(* IEC 61131-3 sources: MotionTestBenchMaster/Logical/30_MC/Task/Cyclic03/MC_INTERFACE, 10 files *)

(* ---- HmiInterfaces.st ---- *)
ACTION HmiInterfaces:
	xAxisInVelocityControl	:= FALSE;

	IF VAR_Machine.iq_stParameter.i_uiAxisSelected >= CST_FillerSubModuleHmiStart AND VAR_Machine.iq_stParameter.i_uiAxisSelected <= CST_FillerSubModuleHmiStart + CST_LastFillerModuleAxis	THEN

		VAR_Machine.stFillerModule.iq_stParameters.i_uiAxisSelected	:= VAR_Machine.iq_stParameter.i_uiAxisSelected - CST_FillerSubModuleHmiStart;

		HMI_MC_GenericAxisData.uiDiagCode				:= VAR_Machine.stFillerModule.iq_astSubModuleAxis[VAR_Machine.stFillerModule.iq_stParameters.i_uiAxisSelected].iq_stStatus.q_stMainAxisStatus.q_stInfo.Diag.StatusID.Code;
		HMI_MC_GenericAxisData.iNextAx_Number;
		HMI_MC_GenericAxisData.iPrevAx_Number;
		HMI_MC_GenericAxisData.rEncoderTemperature		:= VAR_Machine.stFillerModule.iq_astSubModuleAxis[VAR_Machine.stFillerModule.iq_stParameters.i_uiAxisSelected].iq_stStatus.q_stMainAxisStatus.q_rEncoderTemperature;
		HMI_MC_GenericAxisData.rMaxTorque;
		HMI_MC_GenericAxisData.rMotorTemperature		:= VAR_Machine.stFillerModule.iq_astSubModuleAxis[VAR_Machine.stFillerModule.iq_stParameters.i_uiAxisSelected].iq_stStatus.q_stMainAxisStatus.q_rMotorTemperature;
		HMI_MC_GenericAxisData.rNextAx_Position_mm;
		HMI_MC_GenericAxisData.rPosition				:= LREAL_TO_REAL(VAR_Machine.stFillerModule.iq_astSubModuleAxis[VAR_Machine.stFillerModule.iq_stParameters.i_uiAxisSelected].iq_stStatus.q_stMainAxisStatus.q_lrPosition);
		HMI_MC_GenericAxisData.rPosition_mm				:= FC_DegreeToMm(CFG_MC.Mechanical.MachineStep, HMI_MC_GenericAxisData.rPosition, TRUE);

		HMI_MC_GenericAxisData.xMotorWithBrake			:= VAR_Machine.stFillerModule.iq_astSubModuleAxis[VAR_Machine.stFillerModule.iq_stParameters.i_uiAxisSelected].iq_stStatus.q_stMainAxisStatus.q_xMotorWithBrake;
		HMI_MC_GenericAxisData.xThirdPartMotor			:= VAR_Machine.stFillerModule.iq_astSubModuleAxis[VAR_Machine.stFillerModule.iq_stParameters.i_uiAxisSelected].iq_stStatus.q_stMainAxisStatus.q_xThirdPartyMotor;
		HMI_MC_GenericAxisData.xVelocityControl			:= VAR_Machine.stFillerModule.iq_astSubModuleAxis[VAR_Machine.stFillerModule.iq_stParameters.i_uiAxisSelected].iq_stStatus.q_stMainAxisStatus.q_xVelocityControl;
		HMI_MC_GenericAxisData.xInduction				:= VAR_Machine.stFillerModule.iq_astSubModuleAxis[VAR_Machine.stFillerModule.iq_stParameters.i_uiAxisSelected].iq_stStatus.q_stMainAxisStatus.q_xInduction;
		HMI_MC_GenericAxisData.rHomingOffset			:= VAR_Machine.stFillerModule.iq_astSubModuleAxis[VAR_Machine.stFillerModule.iq_stParameters.i_uiAxisSelected].iq_stStatus.q_stMainAxisStatus.q_rHomingOffset;

		HMI_MC_GenericAxisData.rTotalPhasingOffset		:= FC_DegreeToMm(CFG_MC.Mechanical.MachineStep,VAR_Machine.stFillerModule.iq_astSubModuleAxis[VAR_Machine.stFillerModule.iq_stParameters.i_uiAxisSelected].iq_stStatus.q_stMainAxisStatus.q_rTotalOffset, FALSE);

		HMI_MC_GenericAxisData.rLagError				:= FC_DegreeToMm(CFG_MC.Mechanical.MachineStep, VAR_Machine.stFillerModule.iq_astSubModuleAxis[VAR_Machine.stFillerModule.iq_stParameters.i_uiAxisSelected].iq_stStatus.q_stMainAxisStatus.q_rLagError, FALSE);

		HMI_MC_GenericAxisData.rPrevAx_Position_mm;
		HMI_MC_GenericAxisData.rTorque					:= LREAL_TO_REAL(VAR_Machine.stFillerModule.iq_astSubModuleAxis[VAR_Machine.stFillerModule.iq_stParameters.i_uiAxisSelected].iq_stStatus.q_stMainAxisStatus.q_lrTorque);
		HMI_MC_GenericAxisData.rVelocity				:= VAR_Machine.stFillerModule.iq_astSubModuleAxis[VAR_Machine.stFillerModule.iq_stParameters.i_uiAxisSelected].iq_stStatus.q_stMainAxisStatus.q_rVelocity * 10.0;
		HMI_MC_GenericAxisData.rSwitchValue;

		HMI_MC_GenericAxisData.xInitialized				:= VAR_Machine.stFillerModule.iq_astSubModuleAxis[VAR_Machine.stFillerModule.iq_stParameters.i_uiAxisSelected].iq_stStatus.q_stMainAxisStatus.q_xInitDone;

		xPhasingRunning									:= VAR_Machine.stFillerModule.iq_astSubModuleAxis[VAR_Machine.stFillerModule.iq_stParameters.i_uiAxisSelected].iq_stStatus.q_stMainAxisStatus.q_xPhasingRunning;

		IF HMI_MC_GenericAxisData.xInitialized THEN
			HMI_MC_GenericAxisData.xActive				:= VAR_Machine.stFillerModule.iq_astSubModuleAxis[VAR_Machine.stFillerModule.iq_stParameters.i_uiAxisSelected].iq_stStatus.q_stMainAxisStatus.q_xActive;
			HMI_MC_GenericAxisData.xBrakeReleased		:= VAR_Machine.stFillerModule.iq_astSubModuleAxis[VAR_Machine.stFillerModule.iq_stParameters.i_uiAxisSelected].iq_stStatus.q_stMainAxisStatus.q_xBrakeReleased;
			HMI_MC_GenericAxisData.xEnabled;
			HMI_MC_GenericAxisData.xFollowingError		:= VAR_Machine.stFillerModule.iq_astSubModuleAxis[VAR_Machine.stFillerModule.iq_stParameters.i_uiAxisSelected].iq_stStatus.q_stMainAxisStatus.q_xLagError;
			HMI_MC_GenericAxisData.xHomed				:= VAR_Machine.stFillerModule.iq_astSubModuleAxis[VAR_Machine.stFillerModule.iq_stParameters.i_uiAxisSelected].iq_stStatus.q_stMainAxisStatus.q_xIsHomed;
			HMI_MC_GenericAxisData.xInError				:= VAR_Machine.stFillerModule.iq_astSubModuleAxis[VAR_Machine.stFillerModule.iq_stParameters.i_uiAxisSelected].iq_stStatus.q_stMainAxisStatus.q_xError;
			HMI_MC_GenericAxisData.xInPosition			:= VAR_Machine.stFillerModule.iq_astSubModuleAxis[VAR_Machine.stFillerModule.iq_stParameters.i_uiAxisSelected].iq_stStatus.q_stMainAxisStatus.q_xInPosition;
			HMI_MC_GenericAxisData.xPowered				:= VAR_Machine.stFillerModule.iq_astSubModuleAxis[VAR_Machine.stFillerModule.iq_stParameters.i_uiAxisSelected].iq_stStatus.q_stMainAxisStatus.q_xPoweredOn;
			HMI_MC_GenericAxisData.xReal				:= VAR_Machine.stFillerModule.iq_astSubModuleAxis[VAR_Machine.stFillerModule.iq_stParameters.i_uiAxisSelected].iq_stStatus.q_stMainAxisStatus.q_xAxisReal;
			HMI_MC_GenericAxisData.xRunning				:= NOT VAR_Machine.stFillerModule.iq_astSubModuleAxis[VAR_Machine.stFillerModule.iq_stParameters.i_uiAxisSelected].iq_stStatus.q_stMainAxisStatus.q_xStopped;
			HMI_MC_GenericAxisData.xSynchro				:= VAR_Machine.stFillerModule.iq_astSubModuleAxis[VAR_Machine.stFillerModule.iq_stParameters.i_uiAxisSelected].iq_stStatus.q_stMainAxisStatus.q_xSynchronized;
			HMI_MC_GenericAxisData.xTorqueError			:= VAR_Machine.stFillerModule.iq_astSubModuleAxis[VAR_Machine.stFillerModule.iq_stParameters.i_uiAxisSelected].iq_stStatus.q_stMainAxisStatus.q_xTorqueError;
			HMI_MC_GenericAxisData.xHmiWait				:= FALSE;
		ELSE
			HMI_MC_GenericAxisData.xActive				:= FALSE;
			HMI_MC_GenericAxisData.xBrakeReleased		:= FALSE;
			HMI_MC_GenericAxisData.xEnabled;
			HMI_MC_GenericAxisData.xFollowingError		:= FALSE;
			HMI_MC_GenericAxisData.xHomed				:= FALSE;
			HMI_MC_GenericAxisData.xInError				:= FALSE;
			HMI_MC_GenericAxisData.xInPosition			:= FALSE;
			HMI_MC_GenericAxisData.xPowered				:= FALSE;
			HMI_MC_GenericAxisData.xReal				:= FALSE;
			HMI_MC_GenericAxisData.xRunning				:= FALSE;
			HMI_MC_GenericAxisData.xSynchro				:= FALSE;
			HMI_MC_GenericAxisData.xTorqueError			:= FALSE;
			HMI_MC_GenericAxisData.xHmiWait				:= TRUE;
		END_IF

		xAxisInVelocityControl	:= VAR_Machine.stFillerModule.iq_astSubModuleAxis[VAR_Machine.stFillerModule.iq_stParameters.i_uiAxisSelected].iq_stStatus.q_stMainAxisStatus.q_xVelocityControl;

	ELSIF VAR_Machine.iq_stParameter.i_uiAxisSelected >= CST_OutletSubModuleHmiStart AND VAR_Machine.iq_stParameter.i_uiAxisSelected <= CST_OutletSubModuleHmiStart + CST_LastOutletModuleAxis THEN

		VAR_Machine.stOutletModule.iq_stParameters.i_uiAxisSelected	:= VAR_Machine.iq_stParameter.i_uiAxisSelected - CST_OutletSubModuleHmiStart;

		HMI_MC_GenericAxisData.uiDiagCode				:= VAR_Machine.stOutletModule.iq_astSubModuleAxis[VAR_Machine.stOutletModule.iq_stParameters.i_uiAxisSelected].iq_stStatus.q_stMainAxisStatus.q_stInfo.Diag.StatusID.Code;
		HMI_MC_GenericAxisData.iNextAx_Number;
		HMI_MC_GenericAxisData.iPrevAx_Number;
		HMI_MC_GenericAxisData.rEncoderTemperature		:= VAR_Machine.stOutletModule.iq_astSubModuleAxis[VAR_Machine.stOutletModule.iq_stParameters.i_uiAxisSelected].iq_stStatus.q_stMainAxisStatus.q_rEncoderTemperature;
		HMI_MC_GenericAxisData.rMaxTorque;
		HMI_MC_GenericAxisData.rLagError				:= FC_DegreeToMm(CFG_MC.Mechanical.MachineStep, VAR_Machine.stOutletModule.iq_astSubModuleAxis[VAR_Machine.stOutletModule.iq_stParameters.i_uiAxisSelected].iq_stStatus.q_stMainAxisStatus.q_rLagError, FALSE);

		HMI_MC_GenericAxisData.xMotorWithBrake			:= VAR_Machine.stOutletModule.iq_astSubModuleAxis[VAR_Machine.stOutletModule.iq_stParameters.i_uiAxisSelected].iq_stStatus.q_stMainAxisStatus.q_xMotorWithBrake;
		HMI_MC_GenericAxisData.xThirdPartMotor			:= VAR_Machine.stOutletModule.iq_astSubModuleAxis[VAR_Machine.stOutletModule.iq_stParameters.i_uiAxisSelected].iq_stStatus.q_stMainAxisStatus.q_xThirdPartyMotor;
		HMI_MC_GenericAxisData.xVelocityControl			:= VAR_Machine.stOutletModule.iq_astSubModuleAxis[VAR_Machine.stOutletModule.iq_stParameters.i_uiAxisSelected].iq_stStatus.q_stMainAxisStatus.q_xVelocityControl;
		HMI_MC_GenericAxisData.xInduction				:= VAR_Machine.stOutletModule.iq_astSubModuleAxis[VAR_Machine.stOutletModule.iq_stParameters.i_uiAxisSelected].iq_stStatus.q_stMainAxisStatus.q_xInduction;
		HMI_MC_GenericAxisData.rHomingOffset			:= VAR_Machine.stOutletModule.iq_astSubModuleAxis[VAR_Machine.stOutletModule.iq_stParameters.i_uiAxisSelected].iq_stStatus.q_stMainAxisStatus.q_rHomingOffset;

		HMI_MC_GenericAxisData.rMotorTemperature		:= VAR_Machine.stOutletModule.iq_astSubModuleAxis[VAR_Machine.stOutletModule.iq_stParameters.i_uiAxisSelected].iq_stStatus.q_stMainAxisStatus.q_rMotorTemperature;
		HMI_MC_GenericAxisData.rNextAx_Position_mm;
		HMI_MC_GenericAxisData.rPosition				:= LREAL_TO_REAL(VAR_Machine.stOutletModule.iq_astSubModuleAxis[VAR_Machine.stOutletModule.iq_stParameters.i_uiAxisSelected].iq_stStatus.q_stMainAxisStatus.q_lrPosition);
		HMI_MC_GenericAxisData.rPosition_mm				:= FC_DegreeToMm(CFG_MC.Mechanical.MachineStep, HMI_MC_GenericAxisData.rPosition, TRUE);

		HMI_MC_GenericAxisData.rPrevAx_Position_mm;
		HMI_MC_GenericAxisData.rTorque					:= LREAL_TO_REAL(VAR_Machine.stOutletModule.iq_astSubModuleAxis[VAR_Machine.stOutletModule.iq_stParameters.i_uiAxisSelected].iq_stStatus.q_stMainAxisStatus.q_lrTorque);
		HMI_MC_GenericAxisData.rVelocity				:= VAR_Machine.stOutletModule.iq_astSubModuleAxis[VAR_Machine.stOutletModule.iq_stParameters.i_uiAxisSelected].iq_stStatus.q_stMainAxisStatus.q_rVelocity * 10.0;
		HMI_MC_GenericAxisData.rSwitchValue;

		HMI_MC_GenericAxisData.rTotalPhasingOffset		:= FC_DegreeToMm(CFG_MC.Mechanical.MachineStep,VAR_Machine.stOutletModule.iq_astSubModuleAxis[VAR_Machine.stOutletModule.iq_stParameters.i_uiAxisSelected].iq_stStatus.q_stMainAxisStatus.q_rTotalOffset,FALSE);

		HMI_MC_GenericAxisData.xInitialized				:= VAR_Machine.stOutletModule.iq_astSubModuleAxis[VAR_Machine.stOutletModule.iq_stParameters.i_uiAxisSelected].iq_stStatus.q_stMainAxisStatus.q_xInitDone;

		xPhasingRunning									:= VAR_Machine.stOutletModule.iq_astSubModuleAxis[VAR_Machine.stOutletModule.iq_stParameters.i_uiAxisSelected].iq_stStatus.q_stMainAxisStatus.q_xPhasingRunning;

		IF HMI_MC_GenericAxisData.xInitialized THEN
			HMI_MC_GenericAxisData.xActive				:= VAR_Machine.stOutletModule.iq_astSubModuleAxis[VAR_Machine.stOutletModule.iq_stParameters.i_uiAxisSelected].iq_stStatus.q_stMainAxisStatus.q_xActive;
			HMI_MC_GenericAxisData.xBrakeReleased		:= VAR_Machine.stOutletModule.iq_astSubModuleAxis[VAR_Machine.stOutletModule.iq_stParameters.i_uiAxisSelected].iq_stStatus.q_stMainAxisStatus.q_xBrakeReleased;
			HMI_MC_GenericAxisData.xEnabled;
			HMI_MC_GenericAxisData.xFollowingError		:= VAR_Machine.stOutletModule.iq_astSubModuleAxis[VAR_Machine.stOutletModule.iq_stParameters.i_uiAxisSelected].iq_stStatus.q_stMainAxisStatus.q_xLagError;
			HMI_MC_GenericAxisData.xHomed				:= VAR_Machine.stOutletModule.iq_astSubModuleAxis[VAR_Machine.stOutletModule.iq_stParameters.i_uiAxisSelected].iq_stStatus.q_stMainAxisStatus.q_xIsHomed;
			HMI_MC_GenericAxisData.xInError				:= VAR_Machine.stOutletModule.iq_astSubModuleAxis[VAR_Machine.stOutletModule.iq_stParameters.i_uiAxisSelected].iq_stStatus.q_stMainAxisStatus.q_xError;
			HMI_MC_GenericAxisData.xInPosition			:= VAR_Machine.stOutletModule.iq_astSubModuleAxis[VAR_Machine.stOutletModule.iq_stParameters.i_uiAxisSelected].iq_stStatus.q_stMainAxisStatus.q_xInPosition;
			HMI_MC_GenericAxisData.xPowered				:= VAR_Machine.stOutletModule.iq_astSubModuleAxis[VAR_Machine.stOutletModule.iq_stParameters.i_uiAxisSelected].iq_stStatus.q_stMainAxisStatus.q_xPoweredOn;
			HMI_MC_GenericAxisData.xReal				:= VAR_Machine.stOutletModule.iq_astSubModuleAxis[VAR_Machine.stOutletModule.iq_stParameters.i_uiAxisSelected].iq_stStatus.q_stMainAxisStatus.q_xAxisReal;
			HMI_MC_GenericAxisData.xRunning				:= NOT VAR_Machine.stOutletModule.iq_astSubModuleAxis[VAR_Machine.stOutletModule.iq_stParameters.i_uiAxisSelected].iq_stStatus.q_stMainAxisStatus.q_xStopped;
			HMI_MC_GenericAxisData.xSynchro				:= VAR_Machine.stOutletModule.iq_astSubModuleAxis[VAR_Machine.stOutletModule.iq_stParameters.i_uiAxisSelected].iq_stStatus.q_stMainAxisStatus.q_xSynchronized;
			HMI_MC_GenericAxisData.xTorqueError			:= VAR_Machine.stOutletModule.iq_astSubModuleAxis[VAR_Machine.stOutletModule.iq_stParameters.i_uiAxisSelected].iq_stStatus.q_stMainAxisStatus.q_xTorqueError;
			HMI_MC_GenericAxisData.xHmiWait				:= FALSE;
		ELSE
			HMI_MC_GenericAxisData.xActive				:= FALSE;
			HMI_MC_GenericAxisData.xBrakeReleased		:= FALSE;
			HMI_MC_GenericAxisData.xEnabled;
			HMI_MC_GenericAxisData.xFollowingError		:= FALSE;
			HMI_MC_GenericAxisData.xHomed				:= FALSE;
			HMI_MC_GenericAxisData.xInError				:= FALSE;
			HMI_MC_GenericAxisData.xInPosition			:= FALSE;
			HMI_MC_GenericAxisData.xPowered				:= FALSE;
			HMI_MC_GenericAxisData.xReal				:= FALSE;
			HMI_MC_GenericAxisData.xRunning				:= FALSE;
			HMI_MC_GenericAxisData.xSynchro				:= FALSE;
			HMI_MC_GenericAxisData.xTorqueError			:= FALSE;
			HMI_MC_GenericAxisData.xHmiWait				:= TRUE;
		END_IF

		xAxisInVelocityControl	:= VAR_Machine.stOutletModule.iq_astSubModuleAxis[VAR_Machine.stOutletModule.iq_stParameters.i_uiAxisSelected].iq_stStatus.q_stMainAxisStatus.q_xVelocityControl;

	ELSIF VAR_Machine.iq_stParameter.i_uiAxisSelected >= CST_InletSubModuleHmiStart AND VAR_Machine.iq_stParameter.i_uiAxisSelected <= CST_InletSubModuleHmiStart + CST_LastInletModuleAxis THEN

		VAR_Machine.stInletModule.iq_stParameters.i_uiAxisSelected	:= VAR_Machine.iq_stParameter.i_uiAxisSelected - CST_InletSubModuleHmiStart;

		HMI_MC_GenericAxisData.uiDiagCode				:= VAR_Machine.stInletModule.iq_astSubModuleAxis[VAR_Machine.stInletModule.iq_stParameters.i_uiAxisSelected].iq_stStatus.q_stMainAxisStatus.q_stInfo.Diag.StatusID.Code;
		HMI_MC_GenericAxisData.iNextAx_Number;
		HMI_MC_GenericAxisData.iPrevAx_Number;
		HMI_MC_GenericAxisData.rEncoderTemperature		:= VAR_Machine.stInletModule.iq_astSubModuleAxis[VAR_Machine.stInletModule.iq_stParameters.i_uiAxisSelected].iq_stStatus.q_stMainAxisStatus.q_rEncoderTemperature;
		HMI_MC_GenericAxisData.rMaxTorque;
		HMI_MC_GenericAxisData.rLagError				:= FC_DegreeToMm(CFG_MC.Mechanical.MachineStep, VAR_Machine.stInletModule.iq_astSubModuleAxis[VAR_Machine.stInletModule.iq_stParameters.i_uiAxisSelected].iq_stStatus.q_stMainAxisStatus.q_rLagError, FALSE);

		HMI_MC_GenericAxisData.xMotorWithBrake			:= VAR_Machine.stInletModule.iq_astSubModuleAxis[VAR_Machine.stInletModule.iq_stParameters.i_uiAxisSelected].iq_stStatus.q_stMainAxisStatus.q_xMotorWithBrake;
		HMI_MC_GenericAxisData.xThirdPartMotor			:= VAR_Machine.stInletModule.iq_astSubModuleAxis[VAR_Machine.stInletModule.iq_stParameters.i_uiAxisSelected].iq_stStatus.q_stMainAxisStatus.q_xThirdPartyMotor;
		HMI_MC_GenericAxisData.xVelocityControl			:= VAR_Machine.stInletModule.iq_astSubModuleAxis[VAR_Machine.stInletModule.iq_stParameters.i_uiAxisSelected].iq_stStatus.q_stMainAxisStatus.q_xVelocityControl;
		HMI_MC_GenericAxisData.xInduction				:= VAR_Machine.stInletModule.iq_astSubModuleAxis[VAR_Machine.stInletModule.iq_stParameters.i_uiAxisSelected].iq_stStatus.q_stMainAxisStatus.q_xInduction;
		HMI_MC_GenericAxisData.rHomingOffset			:= VAR_Machine.stInletModule.iq_astSubModuleAxis[VAR_Machine.stInletModule.iq_stParameters.i_uiAxisSelected].iq_stStatus.q_stMainAxisStatus.q_rHomingOffset;

		HMI_MC_GenericAxisData.rMotorTemperature		:= VAR_Machine.stInletModule.iq_astSubModuleAxis[VAR_Machine.stInletModule.iq_stParameters.i_uiAxisSelected].iq_stStatus.q_stMainAxisStatus.q_rMotorTemperature;
		HMI_MC_GenericAxisData.rNextAx_Position_mm;
		HMI_MC_GenericAxisData.rPosition				:= LREAL_TO_REAL(VAR_Machine.stInletModule.iq_astSubModuleAxis[VAR_Machine.stInletModule.iq_stParameters.i_uiAxisSelected].iq_stStatus.q_stMainAxisStatus.q_lrPosition);
		HMI_MC_GenericAxisData.rPosition_mm				:= FC_DegreeToMm(CFG_MC.Mechanical.MachineStep, HMI_MC_GenericAxisData.rPosition, TRUE);

		HMI_MC_GenericAxisData.rPrevAx_Position_mm;
		HMI_MC_GenericAxisData.rTorque					:= LREAL_TO_REAL(VAR_Machine.stInletModule.iq_astSubModuleAxis[VAR_Machine.stInletModule.iq_stParameters.i_uiAxisSelected].iq_stStatus.q_stMainAxisStatus.q_lrTorque);
		HMI_MC_GenericAxisData.rVelocity				:= VAR_Machine.stInletModule.iq_astSubModuleAxis[VAR_Machine.stInletModule.iq_stParameters.i_uiAxisSelected].iq_stStatus.q_stMainAxisStatus.q_rVelocity * 10.0;
		HMI_MC_GenericAxisData.rSwitchValue;

		HMI_MC_GenericAxisData.rTotalPhasingOffset		:= FC_DegreeToMm(CFG_MC.Mechanical.MachineStep,VAR_Machine.stInletModule.iq_astSubModuleAxis[VAR_Machine.stInletModule.iq_stParameters.i_uiAxisSelected].iq_stStatus.q_stMainAxisStatus.q_rTotalOffset,FALSE);

		HMI_MC_GenericAxisData.xInitialized				:= VAR_Machine.stInletModule.iq_astSubModuleAxis[VAR_Machine.stInletModule.iq_stParameters.i_uiAxisSelected].iq_stStatus.q_stMainAxisStatus.q_xInitDone;

		xPhasingRunning									:= VAR_Machine.stInletModule.iq_astSubModuleAxis[VAR_Machine.stInletModule.iq_stParameters.i_uiAxisSelected].iq_stStatus.q_stMainAxisStatus.q_xPhasingRunning;

		IF HMI_MC_GenericAxisData.xInitialized THEN
			HMI_MC_GenericAxisData.xActive				:= VAR_Machine.stInletModule.iq_astSubModuleAxis[VAR_Machine.stInletModule.iq_stParameters.i_uiAxisSelected].iq_stStatus.q_stMainAxisStatus.q_xActive;
			HMI_MC_GenericAxisData.xBrakeReleased		:= VAR_Machine.stInletModule.iq_astSubModuleAxis[VAR_Machine.stInletModule.iq_stParameters.i_uiAxisSelected].iq_stStatus.q_stMainAxisStatus.q_xBrakeReleased;
			HMI_MC_GenericAxisData.xEnabled;
			HMI_MC_GenericAxisData.xFollowingError		:= VAR_Machine.stInletModule.iq_astSubModuleAxis[VAR_Machine.stInletModule.iq_stParameters.i_uiAxisSelected].iq_stStatus.q_stMainAxisStatus.q_xLagError;
			HMI_MC_GenericAxisData.xHomed				:= VAR_Machine.stInletModule.iq_astSubModuleAxis[VAR_Machine.stInletModule.iq_stParameters.i_uiAxisSelected].iq_stStatus.q_stMainAxisStatus.q_xIsHomed;
			HMI_MC_GenericAxisData.xInError				:= VAR_Machine.stInletModule.iq_astSubModuleAxis[VAR_Machine.stInletModule.iq_stParameters.i_uiAxisSelected].iq_stStatus.q_stMainAxisStatus.q_xError;
			HMI_MC_GenericAxisData.xInPosition			:= VAR_Machine.stInletModule.iq_astSubModuleAxis[VAR_Machine.stInletModule.iq_stParameters.i_uiAxisSelected].iq_stStatus.q_stMainAxisStatus.q_xInPosition;
			HMI_MC_GenericAxisData.xPowered				:= VAR_Machine.stInletModule.iq_astSubModuleAxis[VAR_Machine.stInletModule.iq_stParameters.i_uiAxisSelected].iq_stStatus.q_stMainAxisStatus.q_xPoweredOn;
			HMI_MC_GenericAxisData.xReal				:= VAR_Machine.stInletModule.iq_astSubModuleAxis[VAR_Machine.stInletModule.iq_stParameters.i_uiAxisSelected].iq_stStatus.q_stMainAxisStatus.q_xAxisReal;
			HMI_MC_GenericAxisData.xRunning				:= NOT VAR_Machine.stInletModule.iq_astSubModuleAxis[VAR_Machine.stInletModule.iq_stParameters.i_uiAxisSelected].iq_stStatus.q_stMainAxisStatus.q_xStopped;
			HMI_MC_GenericAxisData.xSynchro				:= VAR_Machine.stInletModule.iq_astSubModuleAxis[VAR_Machine.stInletModule.iq_stParameters.i_uiAxisSelected].iq_stStatus.q_stMainAxisStatus.q_xSynchronized;
			HMI_MC_GenericAxisData.xTorqueError			:= VAR_Machine.stInletModule.iq_astSubModuleAxis[VAR_Machine.stInletModule.iq_stParameters.i_uiAxisSelected].iq_stStatus.q_stMainAxisStatus.q_xTorqueError;
			HMI_MC_GenericAxisData.xHmiWait				:= FALSE;
		ELSE
			HMI_MC_GenericAxisData.xActive				:= FALSE;
			HMI_MC_GenericAxisData.xBrakeReleased		:= FALSE;
			HMI_MC_GenericAxisData.xEnabled;
			HMI_MC_GenericAxisData.xFollowingError		:= FALSE;
			HMI_MC_GenericAxisData.xHomed				:= FALSE;
			HMI_MC_GenericAxisData.xInError				:= FALSE;
			HMI_MC_GenericAxisData.xInPosition			:= FALSE;
			HMI_MC_GenericAxisData.xPowered				:= FALSE;
			HMI_MC_GenericAxisData.xReal				:= FALSE;
			HMI_MC_GenericAxisData.xRunning				:= FALSE;
			HMI_MC_GenericAxisData.xSynchro				:= FALSE;
			HMI_MC_GenericAxisData.xTorqueError			:= FALSE;
			HMI_MC_GenericAxisData.xHmiWait				:= TRUE;
		END_IF

		xAxisInVelocityControl	:= VAR_Machine.stInletModule.iq_astSubModuleAxis[VAR_Machine.stInletModule.iq_stParameters.i_uiAxisSelected].iq_stStatus.q_stMainAxisStatus.q_xVelocityControl;

	ELSIF VAR_Machine.iq_stParameter.i_uiAxisSelected = CST_MachinePhasingOffset THEN

		VAR_Machine.stMasterModule.iq_stParameters.i_uiAxisSelected	:=	VAR_Machine.iq_stParameter.i_uiAxisSelected;

		HMI_MC_GenericAxisData.uiDiagCode				:= VAR_Machine.stMasterModule.iq_astSubModuleAxis[CST_MachineMasterAxis].iq_stStatus.q_stMainAxisStatus.q_stInfo.Diag.StatusID.Code;
		HMI_MC_GenericAxisData.rLagError				:= FC_DegreeToMm(CFG_MC.Mechanical.MachineStep, VAR_Machine.stMasterModule.iq_astSubModuleAxis[CST_MachineMasterAxis].iq_stStatus.q_stMainAxisStatus.q_rLagError,FALSE);

		HMI_MC_GenericAxisData.xMotorWithBrake			:= VAR_Machine.stMasterModule.iq_astSubModuleAxis[CST_MachineMasterAxis].iq_stStatus.q_stMainAxisStatus.q_xMotorWithBrake;
		HMI_MC_GenericAxisData.xThirdPartMotor			:= VAR_Machine.stMasterModule.iq_astSubModuleAxis[CST_MachineMasterAxis].iq_stStatus.q_stMainAxisStatus.q_xThirdPartyMotor;
		HMI_MC_GenericAxisData.xVelocityControl			:= VAR_Machine.stMasterModule.iq_astSubModuleAxis[CST_MachineMasterAxis].iq_stStatus.q_stMainAxisStatus.q_xVelocityControl;
		HMI_MC_GenericAxisData.xInduction				:= VAR_Machine.stMasterModule.iq_astSubModuleAxis[CST_MachineMasterAxis].iq_stStatus.q_stMainAxisStatus.q_xInduction;
		HMI_MC_GenericAxisData.rHomingOffset			:= VAR_Machine.stMasterModule.iq_astSubModuleAxis[CST_MachineMasterAxis].iq_stStatus.q_stMainAxisStatus.q_rHomingOffset;

		HMI_MC_GenericAxisData.rPosition				:= LREAL_TO_REAL(VAR_Machine.stMasterModule.iq_astSubModuleAxis[CST_MachineMasterAxis].iq_stStatus.q_stMainAxisStatus.q_lrPosition);
		HMI_MC_GenericAxisData.rPosition_mm				:= FC_DegreeToMm(CFG_MC.Mechanical.MachineStep,HMI_MC_GenericAxisData.rPosition,TRUE);

		HMI_MC_GenericAxisData.rVelocity				:= VAR_Machine.stMasterModule.iq_astSubModuleAxis[CST_MachineMasterAxis].iq_stStatus.q_stMainAxisStatus.q_rVelocity * 10.0;

		HMI_MC_GenericAxisData.rTotalPhasingOffset		:= FC_DegreeToMm(CFG_MC.Mechanical.MachineStep,VAR_Machine.stMasterModule.iq_astSubModuleAxis[CST_MachineMasterAxis].iq_stStatus.q_stMainAxisStatus.q_rTotalOffset,FALSE);

		HMI_MC_GenericAxisData.xInitialized				:= VAR_Machine.stMasterModule.iq_astSubModuleAxis[CST_MachineMasterAxis].iq_stStatus.q_stMainAxisStatus.q_xInitDone;

		xPhasingRunning									:= VAR_Machine.stMasterModule.iq_astSubModuleAxis[CST_MachineMasterAxis].iq_stStatus.q_stMainAxisStatus.q_xPhasingRunning;

		IF HMI_MC_GenericAxisData.xInitialized THEN
			HMI_MC_GenericAxisData.xActive				:= VAR_Machine.stMasterModule.iq_astSubModuleAxis[CST_MachineMasterAxis].iq_stStatus.q_stMainAxisStatus.q_xActive;
			HMI_MC_GenericAxisData.xBrakeReleased		:= FALSE;
			HMI_MC_GenericAxisData.xEnabled;
			HMI_MC_GenericAxisData.xFollowingError		:= FALSE;
			HMI_MC_GenericAxisData.xHomed				:= FALSE;
			HMI_MC_GenericAxisData.xInError				:= VAR_Machine.stMasterModule.iq_astSubModuleAxis[CST_MachineMasterAxis].iq_stStatus.q_stMainAxisStatus.q_xError;
			HMI_MC_GenericAxisData.xInPosition			:= VAR_Machine.stMasterModule.iq_astSubModuleAxis[CST_MachineMasterAxis].iq_stStatus.q_stMainAxisStatus.q_xInPosition;
			HMI_MC_GenericAxisData.xPowered				:= FALSE;
			HMI_MC_GenericAxisData.xReal				:= FALSE;
			HMI_MC_GenericAxisData.xRunning				:= FALSE;
			HMI_MC_GenericAxisData.xSynchro				:= VAR_Machine.stMasterModule.iq_astSubModuleAxis[CST_MachineMasterAxis].iq_stStatus.q_stMainAxisStatus.q_xSynchronized;
			HMI_MC_GenericAxisData.xTorqueError			:= FALSE;
			HMI_MC_GenericAxisData.xHmiWait				:= FALSE;
		ELSE
			HMI_MC_GenericAxisData.xActive				:= FALSE;
			HMI_MC_GenericAxisData.xBrakeReleased		:= FALSE;
			HMI_MC_GenericAxisData.xEnabled;
			HMI_MC_GenericAxisData.xFollowingError		:= FALSE;
			HMI_MC_GenericAxisData.xHomed				:= FALSE;
			HMI_MC_GenericAxisData.xInError				:= FALSE;
			HMI_MC_GenericAxisData.xInPosition			:= FALSE;
			HMI_MC_GenericAxisData.xPowered				:= FALSE;
			HMI_MC_GenericAxisData.xReal				:= FALSE;
			HMI_MC_GenericAxisData.xRunning				:= FALSE;
			HMI_MC_GenericAxisData.xSynchro				:= FALSE;
			HMI_MC_GenericAxisData.xTorqueError			:= FALSE;
			HMI_MC_GenericAxisData.xHmiWait				:= TRUE;
		END_IF

		xAxisInVelocityControl	:=	 VAR_Machine.stMasterModule.iq_astSubModuleAxis[CST_MachineMasterAxis].iq_stStatus.q_stMainAxisStatus.q_xVelocityControl;
	END_IF

	CASE VAR_Machine.iq_stParameter.i_uiAxisSelected OF
		99:
			HMI_MC_GenericAxisData.usiHmiName	:= 99; //V4.A.A.1.6.13

		105:
			HMI_MC_GenericAxisData.usiHmiName	:= CFG_MC.Axes.Filler.In[10].HmiNameId;

		106:
			HMI_MC_GenericAxisData.usiHmiName	:= CFG_MC.Axes.Filler.In[9].HmiNameId;

		107:
			HMI_MC_GenericAxisData.usiHmiName	:= CFG_MC.Axes.Filler.In[8].HmiNameId;

		108:
			HMI_MC_GenericAxisData.usiHmiName	:= CFG_MC.Axes.Filler.In[7].HmiNameId;

		109:
			HMI_MC_GenericAxisData.usiHmiName	:= CFG_MC.Axes.Filler.In[6].HmiNameId;

		110:
			HMI_MC_GenericAxisData.usiHmiName	:= CFG_MC.Axes.Filler.In[5].HmiNameId;

		111:
			HMI_MC_GenericAxisData.usiHmiName	:= CFG_MC.Axes.Filler.In[4].HmiNameId;

		112:
			HMI_MC_GenericAxisData.usiHmiName	:= CFG_MC.Axes.Filler.In[3].HmiNameId;

		113:
			HMI_MC_GenericAxisData.usiHmiName	:= CFG_MC.Axes.Filler.In[2].HmiNameId;

		114:
			HMI_MC_GenericAxisData.usiHmiName	:= CFG_MC.Axes.Filler.In[1].HmiNameId;

		115:
			HMI_MC_GenericAxisData.usiHmiName	:= CFG_MC.Axes.Filler.Main.HmiNameId;

		116:
			HMI_MC_GenericAxisData.usiHmiName	:= CFG_MC.Axes.Filler.Out[1].HmiNameId;

		117:
			HMI_MC_GenericAxisData.usiHmiName	:= CFG_MC.Axes.Filler.Out[2].HmiNameId;

		118:
			HMI_MC_GenericAxisData.usiHmiName	:= CFG_MC.Axes.Filler.Out[3].HmiNameId;

		119:
			HMI_MC_GenericAxisData.usiHmiName	:= CFG_MC.Axes.Filler.Out[4].HmiNameId;

		120:
			HMI_MC_GenericAxisData.usiHmiName	:= CFG_MC.Axes.Filler.Out[5].HmiNameId;

		121:
			HMI_MC_GenericAxisData.usiHmiName	:= CFG_MC.Axes.Filler.Out[6].HmiNameId;

		211:
			HMI_MC_GenericAxisData.usiHmiName	:= CFG_MC.Axes.Inlet.In[4].HmiNameId;

		212:
			HMI_MC_GenericAxisData.usiHmiName	:= CFG_MC.Axes.Inlet.In[3].HmiNameId;

		213:
			HMI_MC_GenericAxisData.usiHmiName	:= CFG_MC.Axes.Inlet.In[2].HmiNameId;

		214:
			HMI_MC_GenericAxisData.usiHmiName	:= CFG_MC.Axes.Inlet.In[1].HmiNameId;

		215:
			HMI_MC_GenericAxisData.usiHmiName	:= CFG_MC.Axes.Inlet.Main.HmiNameId;

		216:
			HMI_MC_GenericAxisData.usiHmiName	:= CFG_MC.Axes.Inlet.Out[1].HmiNameId;

		217:
			HMI_MC_GenericAxisData.usiHmiName	:= CFG_MC.Axes.Inlet.Out[2].HmiNameId;

		218:
			HMI_MC_GenericAxisData.usiHmiName	:= CFG_MC.Axes.Inlet.Out[3].HmiNameId;

		219:
			HMI_MC_GenericAxisData.usiHmiName	:= CFG_MC.Axes.Inlet.Out[4].HmiNameId;

		311:
			HMI_MC_GenericAxisData.usiHmiName	:= CFG_MC.Axes.Outlet.In[4].HmiNameId;

		312:
			HMI_MC_GenericAxisData.usiHmiName	:= CFG_MC.Axes.Outlet.In[3].HmiNameId;

		313:
			HMI_MC_GenericAxisData.usiHmiName	:= CFG_MC.Axes.Outlet.In[2].HmiNameId;

		314:
			HMI_MC_GenericAxisData.usiHmiName	:= CFG_MC.Axes.Outlet.In[1].HmiNameId;

		315:
			HMI_MC_GenericAxisData.usiHmiName	:= CFG_MC.Axes.Outlet.Main.HmiNameId;

		316:
			HMI_MC_GenericAxisData.usiHmiName	:= CFG_MC.Axes.Outlet.Out[1].HmiNameId;

		317:
			HMI_MC_GenericAxisData.usiHmiName	:= CFG_MC.Axes.Outlet.Out[2].HmiNameId;

		318:
			HMI_MC_GenericAxisData.usiHmiName	:= CFG_MC.Axes.Outlet.Out[3].HmiNameId;

		319:
			HMI_MC_GenericAxisData.usiHmiName	:= CFG_MC.Axes.Outlet.Out[4].HmiNameId;
		ELSE
			HMI_MC_GenericAxisData.usiHmiName		:= 0;
	END_CASE

	HMI_MC_AxisPresent;

	//Transfer Wheel - Encoder Diagnostic
	HMI_MC_EncoderDiagnostic.Present 	:= CFG_MC.Generic.SyncroPar.ExternalEncoder;
	HMI_MC_EncoderDiagnostic.ModuleOK 	:= MC_InputOutput.Network.Machine.Commands.MasterEncoderPositionValid;
	HMI_MC_EncoderDiagnostic.Value 		:= ITC_Motion_ExtEnc;
END_ACTION

(* ---- HmiInterfacesNew.st ---- *)
ACTION HmiInterfacesNew:
	xAxisInVelocityControl	:= FALSE;

	IF VAR_Machine.iq_stParameter.i_uiAxisSelected >= CST_FillerSubModuleHmiStart AND VAR_Machine.iq_stParameter.i_uiAxisSelected <= CST_FillerSubModuleHmiStart + CST_LastFillerModuleAxis	THEN
		VAR_Machine.stFillerModule.iq_stParameters.i_uiAxisSelected	:= VAR_Machine.iq_stParameter.i_uiAxisSelected - CST_FillerSubModuleHmiStart;
	ELSIF VAR_Machine.iq_stParameter.i_uiAxisSelected >= CST_OutletSubModuleHmiStart AND VAR_Machine.iq_stParameter.i_uiAxisSelected <= CST_OutletSubModuleHmiStart + CST_LastOutletModuleAxis THEN
		VAR_Machine.stOutletModule.iq_stParameters.i_uiAxisSelected	:= VAR_Machine.iq_stParameter.i_uiAxisSelected - CST_OutletSubModuleHmiStart;
	ELSIF VAR_Machine.iq_stParameter.i_uiAxisSelected >= CST_InletSubModuleHmiStart AND VAR_Machine.iq_stParameter.i_uiAxisSelected <= CST_InletSubModuleHmiStart + CST_LastInletModuleAxis THEN
		VAR_Machine.stInletModule.iq_stParameters.i_uiAxisSelected	:= VAR_Machine.iq_stParameter.i_uiAxisSelected - CST_InletSubModuleHmiStart;
	ELSIF VAR_Machine.iq_stParameter.i_uiAxisSelected = CST_MachinePhasingOffset THEN
		VAR_Machine.stMasterModule.iq_stParameters.i_uiAxisSelected	:=	VAR_Machine.iq_stParameter.i_uiAxisSelected;
	END_IF
////////////////////////////////////////////////

		HMI_MC_GenericAxisDataNew[1].uiDiagCode				:= VAR_Machine.stMasterModule.iq_astSubModuleAxis[CST_MachineMasterAxis].iq_stStatus.q_stMainAxisStatus.q_stInfo.Diag.StatusID.Code;
		HMI_MC_GenericAxisDataNew[1].rLagError				:= FC_DegreeToMm(CFG_MC.Mechanical.MachineStep, VAR_Machine.stMasterModule.iq_astSubModuleAxis[CST_MachineMasterAxis].iq_stStatus.q_stMainAxisStatus.q_rLagError,FALSE);

		HMI_MC_GenericAxisDataNew[1].xMotorWithBrake		:= VAR_Machine.stMasterModule.iq_astSubModuleAxis[CST_MachineMasterAxis].iq_stStatus.q_stMainAxisStatus.q_xMotorWithBrake;
		HMI_MC_GenericAxisDataNew[1].xThirdPartMotor		:= VAR_Machine.stMasterModule.iq_astSubModuleAxis[CST_MachineMasterAxis].iq_stStatus.q_stMainAxisStatus.q_xThirdPartyMotor;
		HMI_MC_GenericAxisDataNew[1].xVelocityControl		:= VAR_Machine.stMasterModule.iq_astSubModuleAxis[CST_MachineMasterAxis].iq_stStatus.q_stMainAxisStatus.q_xVelocityControl;
		HMI_MC_GenericAxisDataNew[1].xInduction				:= VAR_Machine.stMasterModule.iq_astSubModuleAxis[CST_MachineMasterAxis].iq_stStatus.q_stMainAxisStatus.q_xInduction;
		HMI_MC_GenericAxisDataNew[1].rHomingOffset			:= VAR_Machine.stMasterModule.iq_astSubModuleAxis[CST_MachineMasterAxis].iq_stStatus.q_stMainAxisStatus.q_rHomingOffset;

		HMI_MC_GenericAxisDataNew[1].rPosition				:= LREAL_TO_REAL(VAR_Machine.stMasterModule.iq_astSubModuleAxis[CST_MachineMasterAxis].iq_stStatus.q_stMainAxisStatus.q_lrPosition);
		HMI_MC_GenericAxisDataNew[1].rPosition_mm			:= FC_DegreeToMm(CFG_MC.Mechanical.MachineStep,HMI_MC_GenericAxisDataNew[1].rPosition,TRUE);//V1.7.2

		HMI_MC_GenericAxisDataNew[1].rVelocity				:= VAR_Machine.stMasterModule.iq_astSubModuleAxis[CST_MachineMasterAxis].iq_stStatus.q_stMainAxisStatus.q_rVelocity * 10.0;

		HMI_MC_GenericAxisDataNew[1].rTotalPhasingOffset	:= FC_DegreeToMm(CFG_MC.Mechanical.MachineStep,VAR_Machine.stMasterModule.iq_astSubModuleAxis[CST_MachineMasterAxis].iq_stStatus.q_stMainAxisStatus.q_rTotalOffset,FALSE);

		HMI_MC_GenericAxisDataNew[1].xInitialized			:= VAR_Machine.stMasterModule.iq_astSubModuleAxis[CST_MachineMasterAxis].iq_stStatus.q_stMainAxisStatus.q_xInitDone;

		xPhasingRunning									:= VAR_Machine.stMasterModule.iq_astSubModuleAxis[CST_MachineMasterAxis].iq_stStatus.q_stMainAxisStatus.q_xPhasingRunning;

		IF HMI_MC_GenericAxisDataNew[1].xInitialized THEN
			HMI_MC_GenericAxisDataNew[1].xActive				:= VAR_Machine.stMasterModule.iq_astSubModuleAxis[CST_MachineMasterAxis].iq_stStatus.q_stMainAxisStatus.q_xActive;
			HMI_MC_GenericAxisDataNew[1].xBrakeReleased		:= FALSE;
			HMI_MC_GenericAxisDataNew[1].xEnabled;
			HMI_MC_GenericAxisDataNew[1].xFollowingError		:= FALSE;
			HMI_MC_GenericAxisDataNew[1].xHomed				:= FALSE;
			HMI_MC_GenericAxisDataNew[1].xInError				:= VAR_Machine.stMasterModule.iq_astSubModuleAxis[CST_MachineMasterAxis].iq_stStatus.q_stMainAxisStatus.q_xError;
			HMI_MC_GenericAxisDataNew[1].xInPosition			:= VAR_Machine.stMasterModule.iq_astSubModuleAxis[CST_MachineMasterAxis].iq_stStatus.q_stMainAxisStatus.q_xInPosition;
			HMI_MC_GenericAxisDataNew[1].xPowered				:= FALSE;
			HMI_MC_GenericAxisDataNew[1].xReal				:= FALSE;
			HMI_MC_GenericAxisDataNew[1].xRunning				:= FALSE;
			HMI_MC_GenericAxisDataNew[1].xSynchro				:= VAR_Machine.stMasterModule.iq_astSubModuleAxis[CST_MachineMasterAxis].iq_stStatus.q_stMainAxisStatus.q_xSynchronized;
			HMI_MC_GenericAxisDataNew[1].xTorqueError			:= FALSE;
//			HMI_MC_GenericAxisDataNew[1].xHmiWait				:= FALSE;//V1.7.2
		ELSE
			HMI_MC_GenericAxisDataNew[1].xActive				:= FALSE;
			HMI_MC_GenericAxisDataNew[1].xBrakeReleased		:= FALSE;
			HMI_MC_GenericAxisDataNew[1].xEnabled;
			HMI_MC_GenericAxisDataNew[1].xFollowingError		:= FALSE;
			HMI_MC_GenericAxisDataNew[1].xHomed				:= FALSE;
			HMI_MC_GenericAxisDataNew[1].xInError				:= FALSE;
			HMI_MC_GenericAxisDataNew[1].xInPosition			:= FALSE;
			HMI_MC_GenericAxisDataNew[1].xPowered				:= FALSE;
			HMI_MC_GenericAxisDataNew[1].xReal				:= FALSE;
			HMI_MC_GenericAxisDataNew[1].xRunning				:= FALSE;
			HMI_MC_GenericAxisDataNew[1].xSynchro				:= FALSE;
			HMI_MC_GenericAxisDataNew[1].xTorqueError			:= FALSE;
//			HMI_MC_GenericAxisDataNew[1].xHmiWait				:= TRUE;//v1.7.2
		END_IF

	FOR HMI_AxisIndex := 1 TO 13 DO
		//Inlet Axis Motor
		IF HMI_MC_GenericAxisDataNew[HMI_AxisIndex].uiAxisID >= CST_InletSubModuleHmiStart AND HMI_MC_GenericAxisDataNew[HMI_AxisIndex].uiAxisID <= CST_InletSubModuleHmiStart + CST_LastInletModuleAxis THEN

			HMI_MC_GenericAxisDataNew[HMI_AxisIndex].uiDiagCode				:= VAR_Machine.stInletModule.iq_astSubModuleAxis[HMI_MC_GenericAxisDataNew[HMI_AxisIndex].uiAxisID-CST_InletSubModuleHmiStart].iq_stStatus.q_stMainAxisStatus.q_stInfo.Diag.StatusID.Code;
			HMI_MC_GenericAxisDataNew[HMI_AxisIndex].iNextAx_Number;
			HMI_MC_GenericAxisDataNew[HMI_AxisIndex].iPrevAx_Number;
			HMI_MC_GenericAxisDataNew[HMI_AxisIndex].rEncoderTemperature		:= VAR_Machine.stInletModule.iq_astSubModuleAxis[HMI_MC_GenericAxisDataNew[HMI_AxisIndex].uiAxisID-CST_InletSubModuleHmiStart].iq_stStatus.q_stMainAxisStatus.q_rEncoderTemperature;
			HMI_MC_GenericAxisDataNew[HMI_AxisIndex].rMaxTorque;
			HMI_MC_GenericAxisDataNew[HMI_AxisIndex].rLagError				:= FC_DegreeToMm(CFG_MC.Mechanical.MachineStep, VAR_Machine.stInletModule.iq_astSubModuleAxis[HMI_MC_GenericAxisDataNew[HMI_AxisIndex].uiAxisID-CST_InletSubModuleHmiStart].iq_stStatus.q_stMainAxisStatus.q_rLagError, FALSE);

			HMI_MC_GenericAxisDataNew[HMI_AxisIndex].xMotorWithBrake			:= VAR_Machine.stInletModule.iq_astSubModuleAxis[HMI_MC_GenericAxisDataNew[HMI_AxisIndex].uiAxisID-CST_InletSubModuleHmiStart].iq_stStatus.q_stMainAxisStatus.q_xMotorWithBrake;
			HMI_MC_GenericAxisDataNew[HMI_AxisIndex].xThirdPartMotor			:= VAR_Machine.stInletModule.iq_astSubModuleAxis[HMI_MC_GenericAxisDataNew[HMI_AxisIndex].uiAxisID-CST_InletSubModuleHmiStart].iq_stStatus.q_stMainAxisStatus.q_xThirdPartyMotor;
			HMI_MC_GenericAxisDataNew[HMI_AxisIndex].xVelocityControl			:= VAR_Machine.stInletModule.iq_astSubModuleAxis[HMI_MC_GenericAxisDataNew[HMI_AxisIndex].uiAxisID-CST_InletSubModuleHmiStart].iq_stStatus.q_stMainAxisStatus.q_xVelocityControl;
			HMI_MC_GenericAxisDataNew[HMI_AxisIndex].xInduction				:= VAR_Machine.stInletModule.iq_astSubModuleAxis[HMI_MC_GenericAxisDataNew[HMI_AxisIndex].uiAxisID-CST_InletSubModuleHmiStart].iq_stStatus.q_stMainAxisStatus.q_xInduction;
			HMI_MC_GenericAxisDataNew[HMI_AxisIndex].rHomingOffset			:= VAR_Machine.stInletModule.iq_astSubModuleAxis[HMI_MC_GenericAxisDataNew[HMI_AxisIndex].uiAxisID-CST_InletSubModuleHmiStart].iq_stStatus.q_stMainAxisStatus.q_rHomingOffset;

			HMI_MC_GenericAxisDataNew[HMI_AxisIndex].rMotorTemperature		:= VAR_Machine.stInletModule.iq_astSubModuleAxis[HMI_MC_GenericAxisDataNew[HMI_AxisIndex].uiAxisID-CST_InletSubModuleHmiStart].iq_stStatus.q_stMainAxisStatus.q_rMotorTemperature;
			HMI_MC_GenericAxisDataNew[HMI_AxisIndex].rNextAx_Position_mm;
			HMI_MC_GenericAxisDataNew[HMI_AxisIndex].rPosition				:= LREAL_TO_REAL(VAR_Machine.stInletModule.iq_astSubModuleAxis[HMI_MC_GenericAxisDataNew[HMI_AxisIndex].uiAxisID-CST_InletSubModuleHmiStart].iq_stStatus.q_stMainAxisStatus.q_lrPosition);
			HMI_MC_GenericAxisDataNew[HMI_AxisIndex].rPosition_mm			:= FC_DegreeToMm(CFG_MC.Mechanical.MachineStep,HMI_MC_GenericAxisDataNew[HMI_AxisIndex].rPosition,TRUE);//v1.7.2

			HMI_MC_GenericAxisDataNew[HMI_AxisIndex].rPrevAx_Position_mm;
			HMI_MC_GenericAxisDataNew[HMI_AxisIndex].rTorque					:= LREAL_TO_REAL(VAR_Machine.stInletModule.iq_astSubModuleAxis[HMI_MC_GenericAxisDataNew[HMI_AxisIndex].uiAxisID-CST_InletSubModuleHmiStart].iq_stStatus.q_stMainAxisStatus.q_lrTorque);
			HMI_MC_GenericAxisDataNew[HMI_AxisIndex].rVelocity				:= VAR_Machine.stInletModule.iq_astSubModuleAxis[HMI_MC_GenericAxisDataNew[HMI_AxisIndex].uiAxisID-CST_InletSubModuleHmiStart].iq_stStatus.q_stMainAxisStatus.q_rVelocity * 10.0;
			HMI_MC_GenericAxisDataNew[HMI_AxisIndex].rSwitchValue;

			HMI_MC_GenericAxisDataNew[HMI_AxisIndex].rTotalPhasingOffset		:= FC_DegreeToMm(CFG_MC.Mechanical.MachineStep,VAR_Machine.stInletModule.iq_astSubModuleAxis[HMI_MC_GenericAxisDataNew[HMI_AxisIndex].uiAxisID-CST_InletSubModuleHmiStart].iq_stStatus.q_stMainAxisStatus.q_rTotalOffset,FALSE);

			HMI_MC_GenericAxisDataNew[HMI_AxisIndex].xInitialized				:= VAR_Machine.stInletModule.iq_astSubModuleAxis[HMI_MC_GenericAxisDataNew[HMI_AxisIndex].uiAxisID-CST_InletSubModuleHmiStart].iq_stStatus.q_stMainAxisStatus.q_xInitDone;

			xPhasingRunning									:= VAR_Machine.stInletModule.iq_astSubModuleAxis[HMI_MC_GenericAxisDataNew[HMI_AxisIndex].uiAxisID-CST_InletSubModuleHmiStart].iq_stStatus.q_stMainAxisStatus.q_xPhasingRunning;

			IF HMI_MC_GenericAxisDataNew[HMI_AxisIndex].xInitialized THEN
				HMI_MC_GenericAxisDataNew[HMI_AxisIndex].xActive				:= VAR_Machine.stInletModule.iq_astSubModuleAxis[HMI_MC_GenericAxisDataNew[HMI_AxisIndex].uiAxisID-CST_InletSubModuleHmiStart].iq_stStatus.q_stMainAxisStatus.q_xActive;
				HMI_MC_GenericAxisDataNew[HMI_AxisIndex].xBrakeReleased		:= VAR_Machine.stInletModule.iq_astSubModuleAxis[HMI_MC_GenericAxisDataNew[HMI_AxisIndex].uiAxisID-CST_InletSubModuleHmiStart].iq_stStatus.q_stMainAxisStatus.q_xBrakeReleased;
				HMI_MC_GenericAxisDataNew[HMI_AxisIndex].xEnabled;
				HMI_MC_GenericAxisDataNew[HMI_AxisIndex].xFollowingError		:= VAR_Machine.stInletModule.iq_astSubModuleAxis[HMI_MC_GenericAxisDataNew[HMI_AxisIndex].uiAxisID-CST_InletSubModuleHmiStart].iq_stStatus.q_stMainAxisStatus.q_xLagError;
				HMI_MC_GenericAxisDataNew[HMI_AxisIndex].xHomed				:= VAR_Machine.stInletModule.iq_astSubModuleAxis[HMI_MC_GenericAxisDataNew[HMI_AxisIndex].uiAxisID-CST_InletSubModuleHmiStart].iq_stStatus.q_stMainAxisStatus.q_xIsHomed;
				HMI_MC_GenericAxisDataNew[HMI_AxisIndex].xInError				:= VAR_Machine.stInletModule.iq_astSubModuleAxis[HMI_MC_GenericAxisDataNew[HMI_AxisIndex].uiAxisID-CST_InletSubModuleHmiStart].iq_stStatus.q_stMainAxisStatus.q_xError;
				HMI_MC_GenericAxisDataNew[HMI_AxisIndex].xInPosition			:= VAR_Machine.stInletModule.iq_astSubModuleAxis[HMI_MC_GenericAxisDataNew[HMI_AxisIndex].uiAxisID-CST_InletSubModuleHmiStart].iq_stStatus.q_stMainAxisStatus.q_xInPosition;
				HMI_MC_GenericAxisDataNew[HMI_AxisIndex].xPowered				:= VAR_Machine.stInletModule.iq_astSubModuleAxis[HMI_MC_GenericAxisDataNew[HMI_AxisIndex].uiAxisID-CST_InletSubModuleHmiStart].iq_stStatus.q_stMainAxisStatus.q_xPoweredOn;
				HMI_MC_GenericAxisDataNew[HMI_AxisIndex].xReal				:= VAR_Machine.stInletModule.iq_astSubModuleAxis[HMI_MC_GenericAxisDataNew[HMI_AxisIndex].uiAxisID-CST_InletSubModuleHmiStart].iq_stStatus.q_stMainAxisStatus.q_xAxisReal;
				HMI_MC_GenericAxisDataNew[HMI_AxisIndex].xRunning				:= NOT VAR_Machine.stInletModule.iq_astSubModuleAxis[HMI_MC_GenericAxisDataNew[HMI_AxisIndex].uiAxisID-CST_InletSubModuleHmiStart].iq_stStatus.q_stMainAxisStatus.q_xStopped;
				HMI_MC_GenericAxisDataNew[HMI_AxisIndex].xSynchro				:= VAR_Machine.stInletModule.iq_astSubModuleAxis[HMI_MC_GenericAxisDataNew[HMI_AxisIndex].uiAxisID-CST_InletSubModuleHmiStart].iq_stStatus.q_stMainAxisStatus.q_xSynchronized;
				HMI_MC_GenericAxisDataNew[HMI_AxisIndex].xTorqueError			:= VAR_Machine.stInletModule.iq_astSubModuleAxis[HMI_MC_GenericAxisDataNew[HMI_AxisIndex].uiAxisID-CST_InletSubModuleHmiStart].iq_stStatus.q_stMainAxisStatus.q_xTorqueError;
				//HMI_MC_GenericAxisDataNew[HMI_AxisIndex].xHmiWait				:= FALSE;//v1.7.2
			ELSE
				HMI_MC_GenericAxisDataNew[HMI_AxisIndex].xActive				:= FALSE;
				HMI_MC_GenericAxisDataNew[HMI_AxisIndex].xBrakeReleased		:= FALSE;
				HMI_MC_GenericAxisDataNew[HMI_AxisIndex].xEnabled;
				HMI_MC_GenericAxisDataNew[HMI_AxisIndex].xFollowingError		:= FALSE;
				HMI_MC_GenericAxisDataNew[HMI_AxisIndex].xHomed					:= FALSE;
				HMI_MC_GenericAxisDataNew[HMI_AxisIndex].xInError				:= FALSE;
				HMI_MC_GenericAxisDataNew[HMI_AxisIndex].xInPosition			:= FALSE;
				HMI_MC_GenericAxisDataNew[HMI_AxisIndex].xPowered				:= FALSE;
				HMI_MC_GenericAxisDataNew[HMI_AxisIndex].xReal					:= FALSE;
				HMI_MC_GenericAxisDataNew[HMI_AxisIndex].xRunning				:= FALSE;
				HMI_MC_GenericAxisDataNew[HMI_AxisIndex].xSynchro				:= FALSE;
				HMI_MC_GenericAxisDataNew[HMI_AxisIndex].xTorqueError			:= FALSE;
//				HMI_MC_GenericAxisDataNew[HMI_AxisIndex].xHmiWait				:= TRUE;//v1.7.2
			END_IF
			xAxisInVelocityControl	:= VAR_Machine.stInletModule.iq_astSubModuleAxis[HMI_MC_GenericAxisDataNew[HMI_AxisIndex].uiAxisID-CST_InletSubModuleHmiStart].iq_stStatus.q_stMainAxisStatus.q_xVelocityControl;
		//Filler Module
		ELSIF HMI_MC_GenericAxisDataNew[HMI_AxisIndex].uiAxisID >= CST_FillerSubModuleHmiStart AND HMI_MC_GenericAxisDataNew[HMI_AxisIndex].uiAxisID <= CST_FillerSubModuleHmiStart + CST_LastFillerModuleAxis THEN
			HMI_MC_GenericAxisDataNew[HMI_AxisIndex].uiDiagCode				:= VAR_Machine.stFillerModule.iq_astSubModuleAxis[HMI_MC_GenericAxisDataNew[HMI_AxisIndex].uiAxisID-CST_FillerSubModuleHmiStart].iq_stStatus.q_stMainAxisStatus.q_stInfo.Diag.StatusID.Code;
			HMI_MC_GenericAxisDataNew[HMI_AxisIndex].iNextAx_Number;
			HMI_MC_GenericAxisDataNew[HMI_AxisIndex].iPrevAx_Number;
			HMI_MC_GenericAxisDataNew[HMI_AxisIndex].rEncoderTemperature		:= VAR_Machine.stFillerModule.iq_astSubModuleAxis[HMI_MC_GenericAxisDataNew[HMI_AxisIndex].uiAxisID-CST_FillerSubModuleHmiStart].iq_stStatus.q_stMainAxisStatus.q_rEncoderTemperature;
			HMI_MC_GenericAxisDataNew[HMI_AxisIndex].rMaxTorque;
			HMI_MC_GenericAxisDataNew[HMI_AxisIndex].rMotorTemperature		:= VAR_Machine.stFillerModule.iq_astSubModuleAxis[HMI_MC_GenericAxisDataNew[HMI_AxisIndex].uiAxisID-CST_FillerSubModuleHmiStart].iq_stStatus.q_stMainAxisStatus.q_rMotorTemperature;
			HMI_MC_GenericAxisDataNew[HMI_AxisIndex].rNextAx_Position_mm;
			HMI_MC_GenericAxisDataNew[HMI_AxisIndex].rPosition				:= LREAL_TO_REAL(VAR_Machine.stFillerModule.iq_astSubModuleAxis[HMI_MC_GenericAxisDataNew[HMI_AxisIndex].uiAxisID-CST_FillerSubModuleHmiStart].iq_stStatus.q_stMainAxisStatus.q_lrPosition);
			HMI_MC_GenericAxisDataNew[HMI_AxisIndex].rPosition_mm			:= FC_DegreeToMm(CFG_MC.Mechanical.MachineStep,HMI_MC_GenericAxisDataNew[HMI_AxisIndex].rPosition,TRUE);//v1.7.2

			HMI_MC_GenericAxisDataNew[HMI_AxisIndex].xMotorWithBrake			:= VAR_Machine.stFillerModule.iq_astSubModuleAxis[HMI_MC_GenericAxisDataNew[HMI_AxisIndex].uiAxisID-CST_FillerSubModuleHmiStart].iq_stStatus.q_stMainAxisStatus.q_xMotorWithBrake;
			HMI_MC_GenericAxisDataNew[HMI_AxisIndex].xThirdPartMotor			:= VAR_Machine.stFillerModule.iq_astSubModuleAxis[HMI_MC_GenericAxisDataNew[HMI_AxisIndex].uiAxisID-CST_FillerSubModuleHmiStart].iq_stStatus.q_stMainAxisStatus.q_xThirdPartyMotor;
			HMI_MC_GenericAxisDataNew[HMI_AxisIndex].xVelocityControl			:= VAR_Machine.stFillerModule.iq_astSubModuleAxis[HMI_MC_GenericAxisDataNew[HMI_AxisIndex].uiAxisID-CST_FillerSubModuleHmiStart].iq_stStatus.q_stMainAxisStatus.q_xVelocityControl;
			HMI_MC_GenericAxisDataNew[HMI_AxisIndex].xInduction				:= VAR_Machine.stFillerModule.iq_astSubModuleAxis[HMI_MC_GenericAxisDataNew[HMI_AxisIndex].uiAxisID-CST_FillerSubModuleHmiStart].iq_stStatus.q_stMainAxisStatus.q_xInduction;
			HMI_MC_GenericAxisDataNew[HMI_AxisIndex].rHomingOffset			:= VAR_Machine.stFillerModule.iq_astSubModuleAxis[HMI_MC_GenericAxisDataNew[HMI_AxisIndex].uiAxisID-CST_FillerSubModuleHmiStart].iq_stStatus.q_stMainAxisStatus.q_rHomingOffset;

			HMI_MC_GenericAxisDataNew[HMI_AxisIndex].rTotalPhasingOffset		:= FC_DegreeToMm(CFG_MC.Mechanical.MachineStep,VAR_Machine.stFillerModule.iq_astSubModuleAxis[HMI_MC_GenericAxisDataNew[HMI_AxisIndex].uiAxisID-CST_FillerSubModuleHmiStart].iq_stStatus.q_stMainAxisStatus.q_rTotalOffset, FALSE);

			HMI_MC_GenericAxisDataNew[HMI_AxisIndex].rLagError				:= FC_DegreeToMm(CFG_MC.Mechanical.MachineStep, VAR_Machine.stFillerModule.iq_astSubModuleAxis[HMI_MC_GenericAxisDataNew[HMI_AxisIndex].uiAxisID-CST_FillerSubModuleHmiStart].iq_stStatus.q_stMainAxisStatus.q_rLagError, FALSE);

			HMI_MC_GenericAxisDataNew[HMI_AxisIndex].rPrevAx_Position_mm;
			HMI_MC_GenericAxisDataNew[HMI_AxisIndex].rTorque					:= LREAL_TO_REAL(VAR_Machine.stFillerModule.iq_astSubModuleAxis[HMI_MC_GenericAxisDataNew[HMI_AxisIndex].uiAxisID-CST_FillerSubModuleHmiStart].iq_stStatus.q_stMainAxisStatus.q_lrTorque);
			HMI_MC_GenericAxisDataNew[HMI_AxisIndex].rVelocity				:= VAR_Machine.stFillerModule.iq_astSubModuleAxis[HMI_MC_GenericAxisDataNew[HMI_AxisIndex].uiAxisID-CST_FillerSubModuleHmiStart].iq_stStatus.q_stMainAxisStatus.q_rVelocity * 10.0;
			HMI_MC_GenericAxisDataNew[HMI_AxisIndex].rSwitchValue;

			HMI_MC_GenericAxisDataNew[HMI_AxisIndex].xInitialized				:= VAR_Machine.stFillerModule.iq_astSubModuleAxis[HMI_MC_GenericAxisDataNew[HMI_AxisIndex].uiAxisID-CST_FillerSubModuleHmiStart].iq_stStatus.q_stMainAxisStatus.q_xInitDone;

			xPhasingRunning									:= VAR_Machine.stFillerModule.iq_astSubModuleAxis[HMI_MC_GenericAxisDataNew[HMI_AxisIndex].uiAxisID-CST_FillerSubModuleHmiStart].iq_stStatus.q_stMainAxisStatus.q_xPhasingRunning;

			IF HMI_MC_GenericAxisDataNew[HMI_AxisIndex].xInitialized THEN
				HMI_MC_GenericAxisDataNew[HMI_AxisIndex].xActive				:= VAR_Machine.stFillerModule.iq_astSubModuleAxis[HMI_MC_GenericAxisDataNew[HMI_AxisIndex].uiAxisID-CST_FillerSubModuleHmiStart].iq_stStatus.q_stMainAxisStatus.q_xActive;
				HMI_MC_GenericAxisDataNew[HMI_AxisIndex].xBrakeReleased		:= VAR_Machine.stFillerModule.iq_astSubModuleAxis[HMI_MC_GenericAxisDataNew[HMI_AxisIndex].uiAxisID-CST_FillerSubModuleHmiStart].iq_stStatus.q_stMainAxisStatus.q_xBrakeReleased;
				HMI_MC_GenericAxisDataNew[HMI_AxisIndex].xEnabled;
				HMI_MC_GenericAxisDataNew[HMI_AxisIndex].xFollowingError		:= VAR_Machine.stFillerModule.iq_astSubModuleAxis[HMI_MC_GenericAxisDataNew[HMI_AxisIndex].uiAxisID-CST_FillerSubModuleHmiStart].iq_stStatus.q_stMainAxisStatus.q_xLagError;
				HMI_MC_GenericAxisDataNew[HMI_AxisIndex].xHomed				:= VAR_Machine.stFillerModule.iq_astSubModuleAxis[HMI_MC_GenericAxisDataNew[HMI_AxisIndex].uiAxisID-CST_FillerSubModuleHmiStart].iq_stStatus.q_stMainAxisStatus.q_xIsHomed;
				HMI_MC_GenericAxisDataNew[HMI_AxisIndex].xInError				:= VAR_Machine.stFillerModule.iq_astSubModuleAxis[HMI_MC_GenericAxisDataNew[HMI_AxisIndex].uiAxisID-CST_FillerSubModuleHmiStart].iq_stStatus.q_stMainAxisStatus.q_xError;
				HMI_MC_GenericAxisDataNew[HMI_AxisIndex].xInPosition			:= VAR_Machine.stFillerModule.iq_astSubModuleAxis[HMI_MC_GenericAxisDataNew[HMI_AxisIndex].uiAxisID-CST_FillerSubModuleHmiStart].iq_stStatus.q_stMainAxisStatus.q_xInPosition;
				HMI_MC_GenericAxisDataNew[HMI_AxisIndex].xPowered				:= VAR_Machine.stFillerModule.iq_astSubModuleAxis[HMI_MC_GenericAxisDataNew[HMI_AxisIndex].uiAxisID-CST_FillerSubModuleHmiStart].iq_stStatus.q_stMainAxisStatus.q_xPoweredOn;
				HMI_MC_GenericAxisDataNew[HMI_AxisIndex].xReal				:= VAR_Machine.stFillerModule.iq_astSubModuleAxis[HMI_MC_GenericAxisDataNew[HMI_AxisIndex].uiAxisID-CST_FillerSubModuleHmiStart].iq_stStatus.q_stMainAxisStatus.q_xAxisReal;
				HMI_MC_GenericAxisDataNew[HMI_AxisIndex].xRunning				:= NOT VAR_Machine.stFillerModule.iq_astSubModuleAxis[HMI_MC_GenericAxisDataNew[HMI_AxisIndex].uiAxisID-CST_FillerSubModuleHmiStart].iq_stStatus.q_stMainAxisStatus.q_xStopped;
				HMI_MC_GenericAxisDataNew[HMI_AxisIndex].xSynchro				:= VAR_Machine.stFillerModule.iq_astSubModuleAxis[HMI_MC_GenericAxisDataNew[HMI_AxisIndex].uiAxisID-CST_FillerSubModuleHmiStart].iq_stStatus.q_stMainAxisStatus.q_xSynchronized;
				HMI_MC_GenericAxisDataNew[HMI_AxisIndex].xTorqueError			:= VAR_Machine.stFillerModule.iq_astSubModuleAxis[HMI_MC_GenericAxisDataNew[HMI_AxisIndex].uiAxisID-CST_FillerSubModuleHmiStart].iq_stStatus.q_stMainAxisStatus.q_xTorqueError;
				//HMI_MC_GenericAxisDataNew[HMI_AxisIndex].xHmiWait				:= FALSE;//v1.7.2
			ELSE
				HMI_MC_GenericAxisDataNew[HMI_AxisIndex].xActive				:= FALSE;
				HMI_MC_GenericAxisDataNew[HMI_AxisIndex].xBrakeReleased		:= FALSE;
				HMI_MC_GenericAxisDataNew[HMI_AxisIndex].xEnabled;
				HMI_MC_GenericAxisDataNew[HMI_AxisIndex].xFollowingError		:= FALSE;
				HMI_MC_GenericAxisDataNew[HMI_AxisIndex].xHomed				:= FALSE;
				HMI_MC_GenericAxisDataNew[HMI_AxisIndex].xInError				:= FALSE;
				HMI_MC_GenericAxisDataNew[HMI_AxisIndex].xInPosition			:= FALSE;
				HMI_MC_GenericAxisDataNew[HMI_AxisIndex].xPowered				:= FALSE;
				HMI_MC_GenericAxisDataNew[HMI_AxisIndex].xReal				:= FALSE;
				HMI_MC_GenericAxisDataNew[HMI_AxisIndex].xRunning				:= FALSE;
				HMI_MC_GenericAxisDataNew[HMI_AxisIndex].xSynchro				:= FALSE;
				HMI_MC_GenericAxisDataNew[HMI_AxisIndex].xTorqueError			:= FALSE;
				//HMI_MC_GenericAxisDataNew[HMI_AxisIndex].xHmiWait				:= TRUE;//v1.7.2
			END_IF

			xAxisInVelocityControl	:= VAR_Machine.stFillerModule.iq_astSubModuleAxis[HMI_MC_GenericAxisDataNew[HMI_AxisIndex].uiAxisID-CST_FillerSubModuleHmiStart].iq_stStatus.q_stMainAxisStatus.q_xVelocityControl;
		//Outlet Module
		ELSIF HMI_MC_GenericAxisDataNew[HMI_AxisIndex].uiAxisID >= CST_OutletSubModuleHmiStart AND HMI_MC_GenericAxisDataNew[HMI_AxisIndex].uiAxisID <= CST_OutletSubModuleHmiStart + CST_LastOutletModuleAxis THEN
			HMI_MC_GenericAxisDataNew[HMI_AxisIndex].uiDiagCode					:= VAR_Machine.stOutletModule.iq_astSubModuleAxis[HMI_MC_GenericAxisDataNew[HMI_AxisIndex].uiAxisID - CST_OutletSubModuleHmiStart].iq_stStatus.q_stMainAxisStatus.q_stInfo.Diag.StatusID.Code;
			HMI_MC_GenericAxisDataNew[HMI_AxisIndex].iNextAx_Number;
			HMI_MC_GenericAxisDataNew[HMI_AxisIndex].iPrevAx_Number;
			HMI_MC_GenericAxisDataNew[HMI_AxisIndex].rEncoderTemperature		:= VAR_Machine.stOutletModule.iq_astSubModuleAxis[HMI_MC_GenericAxisDataNew[HMI_AxisIndex].uiAxisID - CST_OutletSubModuleHmiStart].iq_stStatus.q_stMainAxisStatus.q_rEncoderTemperature;
			HMI_MC_GenericAxisDataNew[HMI_AxisIndex].rMaxTorque;
			HMI_MC_GenericAxisDataNew[HMI_AxisIndex].rLagError					:= FC_DegreeToMm(CFG_MC.Mechanical.MachineStep, VAR_Machine.stOutletModule.iq_astSubModuleAxis[HMI_MC_GenericAxisDataNew[HMI_AxisIndex].uiAxisID - CST_OutletSubModuleHmiStart].iq_stStatus.q_stMainAxisStatus.q_rLagError, FALSE);

			HMI_MC_GenericAxisDataNew[HMI_AxisIndex].xMotorWithBrake			:= VAR_Machine.stOutletModule.iq_astSubModuleAxis[HMI_MC_GenericAxisDataNew[HMI_AxisIndex].uiAxisID - CST_OutletSubModuleHmiStart].iq_stStatus.q_stMainAxisStatus.q_xMotorWithBrake;
			HMI_MC_GenericAxisDataNew[HMI_AxisIndex].xThirdPartMotor			:= VAR_Machine.stOutletModule.iq_astSubModuleAxis[HMI_MC_GenericAxisDataNew[HMI_AxisIndex].uiAxisID - CST_OutletSubModuleHmiStart].iq_stStatus.q_stMainAxisStatus.q_xThirdPartyMotor;
			HMI_MC_GenericAxisDataNew[HMI_AxisIndex].xVelocityControl			:= VAR_Machine.stOutletModule.iq_astSubModuleAxis[HMI_MC_GenericAxisDataNew[HMI_AxisIndex].uiAxisID - CST_OutletSubModuleHmiStart].iq_stStatus.q_stMainAxisStatus.q_xVelocityControl;
			HMI_MC_GenericAxisDataNew[HMI_AxisIndex].xInduction					:= VAR_Machine.stOutletModule.iq_astSubModuleAxis[HMI_MC_GenericAxisDataNew[HMI_AxisIndex].uiAxisID - CST_OutletSubModuleHmiStart].iq_stStatus.q_stMainAxisStatus.q_xInduction;
			HMI_MC_GenericAxisDataNew[HMI_AxisIndex].rHomingOffset				:= VAR_Machine.stOutletModule.iq_astSubModuleAxis[HMI_MC_GenericAxisDataNew[HMI_AxisIndex].uiAxisID - CST_OutletSubModuleHmiStart].iq_stStatus.q_stMainAxisStatus.q_rHomingOffset;

			HMI_MC_GenericAxisDataNew[HMI_AxisIndex].rMotorTemperature			:= VAR_Machine.stOutletModule.iq_astSubModuleAxis[HMI_MC_GenericAxisDataNew[HMI_AxisIndex].uiAxisID - CST_OutletSubModuleHmiStart].iq_stStatus.q_stMainAxisStatus.q_rMotorTemperature;
			HMI_MC_GenericAxisDataNew[HMI_AxisIndex].rNextAx_Position_mm;
			HMI_MC_GenericAxisDataNew[HMI_AxisIndex].rPosition					:= LREAL_TO_REAL(VAR_Machine.stOutletModule.iq_astSubModuleAxis[HMI_MC_GenericAxisDataNew[HMI_AxisIndex].uiAxisID - CST_OutletSubModuleHmiStart].iq_stStatus.q_stMainAxisStatus.q_lrPosition);
			HMI_MC_GenericAxisDataNew[HMI_AxisIndex].rPosition_mm				:= FC_DegreeToMm(CFG_MC.Mechanical.MachineStep,HMI_MC_GenericAxisDataNew[HMI_AxisIndex].rPosition,TRUE);//v1.7.2

			HMI_MC_GenericAxisDataNew[HMI_AxisIndex].rPrevAx_Position_mm;
			HMI_MC_GenericAxisDataNew[HMI_AxisIndex].rTorque					:= LREAL_TO_REAL(VAR_Machine.stOutletModule.iq_astSubModuleAxis[HMI_MC_GenericAxisDataNew[HMI_AxisIndex].uiAxisID - CST_OutletSubModuleHmiStart].iq_stStatus.q_stMainAxisStatus.q_lrTorque);
			HMI_MC_GenericAxisDataNew[HMI_AxisIndex].rVelocity					:= VAR_Machine.stOutletModule.iq_astSubModuleAxis[HMI_MC_GenericAxisDataNew[HMI_AxisIndex].uiAxisID - CST_OutletSubModuleHmiStart].iq_stStatus.q_stMainAxisStatus.q_rVelocity * 10.0;
			HMI_MC_GenericAxisDataNew[HMI_AxisIndex].rSwitchValue;

			HMI_MC_GenericAxisDataNew[HMI_AxisIndex].rTotalPhasingOffset		:= FC_DegreeToMm(CFG_MC.Mechanical.MachineStep,VAR_Machine.stOutletModule.iq_astSubModuleAxis[HMI_MC_GenericAxisDataNew[HMI_AxisIndex].uiAxisID - CST_OutletSubModuleHmiStart].iq_stStatus.q_stMainAxisStatus.q_rTotalOffset,FALSE);

			HMI_MC_GenericAxisDataNew[HMI_AxisIndex].xInitialized				:= VAR_Machine.stOutletModule.iq_astSubModuleAxis[HMI_MC_GenericAxisDataNew[HMI_AxisIndex].uiAxisID - CST_OutletSubModuleHmiStart].iq_stStatus.q_stMainAxisStatus.q_xInitDone;

			xPhasingRunning														:= VAR_Machine.stOutletModule.iq_astSubModuleAxis[HMI_MC_GenericAxisDataNew[HMI_AxisIndex].uiAxisID - CST_OutletSubModuleHmiStart].iq_stStatus.q_stMainAxisStatus.q_xPhasingRunning;

		IF HMI_MC_GenericAxisDataNew[HMI_AxisIndex].xInitialized THEN
			HMI_MC_GenericAxisDataNew[HMI_AxisIndex].xActive				:= VAR_Machine.stOutletModule.iq_astSubModuleAxis[HMI_MC_GenericAxisDataNew[HMI_AxisIndex].uiAxisID - CST_OutletSubModuleHmiStart].iq_stStatus.q_stMainAxisStatus.q_xActive;
			HMI_MC_GenericAxisDataNew[HMI_AxisIndex].xBrakeReleased			:= VAR_Machine.stOutletModule.iq_astSubModuleAxis[HMI_MC_GenericAxisDataNew[HMI_AxisIndex].uiAxisID - CST_OutletSubModuleHmiStart].iq_stStatus.q_stMainAxisStatus.q_xBrakeReleased;
			HMI_MC_GenericAxisDataNew[HMI_AxisIndex].xEnabled;
			HMI_MC_GenericAxisDataNew[HMI_AxisIndex].xFollowingError		:= VAR_Machine.stOutletModule.iq_astSubModuleAxis[HMI_MC_GenericAxisDataNew[HMI_AxisIndex].uiAxisID - CST_OutletSubModuleHmiStart].iq_stStatus.q_stMainAxisStatus.q_xLagError;
			HMI_MC_GenericAxisDataNew[HMI_AxisIndex].xHomed					:= VAR_Machine.stOutletModule.iq_astSubModuleAxis[HMI_MC_GenericAxisDataNew[HMI_AxisIndex].uiAxisID - CST_OutletSubModuleHmiStart].iq_stStatus.q_stMainAxisStatus.q_xIsHomed;
			HMI_MC_GenericAxisDataNew[HMI_AxisIndex].xInError				:= VAR_Machine.stOutletModule.iq_astSubModuleAxis[HMI_MC_GenericAxisDataNew[HMI_AxisIndex].uiAxisID - CST_OutletSubModuleHmiStart].iq_stStatus.q_stMainAxisStatus.q_xError;
			HMI_MC_GenericAxisDataNew[HMI_AxisIndex].xInPosition			:= VAR_Machine.stOutletModule.iq_astSubModuleAxis[HMI_MC_GenericAxisDataNew[HMI_AxisIndex].uiAxisID - CST_OutletSubModuleHmiStart].iq_stStatus.q_stMainAxisStatus.q_xInPosition;
			HMI_MC_GenericAxisDataNew[HMI_AxisIndex].xPowered				:= VAR_Machine.stOutletModule.iq_astSubModuleAxis[HMI_MC_GenericAxisDataNew[HMI_AxisIndex].uiAxisID - CST_OutletSubModuleHmiStart].iq_stStatus.q_stMainAxisStatus.q_xPoweredOn;
			HMI_MC_GenericAxisDataNew[HMI_AxisIndex].xReal					:= VAR_Machine.stOutletModule.iq_astSubModuleAxis[HMI_MC_GenericAxisDataNew[HMI_AxisIndex].uiAxisID - CST_OutletSubModuleHmiStart].iq_stStatus.q_stMainAxisStatus.q_xAxisReal;
			HMI_MC_GenericAxisDataNew[HMI_AxisIndex].xRunning				:= NOT VAR_Machine.stOutletModule.iq_astSubModuleAxis[HMI_MC_GenericAxisDataNew[HMI_AxisIndex].uiAxisID - CST_OutletSubModuleHmiStart].iq_stStatus.q_stMainAxisStatus.q_xStopped;
			HMI_MC_GenericAxisDataNew[HMI_AxisIndex].xSynchro				:= VAR_Machine.stOutletModule.iq_astSubModuleAxis[HMI_MC_GenericAxisDataNew[HMI_AxisIndex].uiAxisID - CST_OutletSubModuleHmiStart].iq_stStatus.q_stMainAxisStatus.q_xSynchronized;
			HMI_MC_GenericAxisDataNew[HMI_AxisIndex].xTorqueError			:= VAR_Machine.stOutletModule.iq_astSubModuleAxis[HMI_MC_GenericAxisDataNew[HMI_AxisIndex].uiAxisID - CST_OutletSubModuleHmiStart].iq_stStatus.q_stMainAxisStatus.q_xTorqueError;
			//HMI_MC_GenericAxisDataNew[HMI_AxisIndex].xHmiWait				:= FALSE;
			ELSE
			HMI_MC_GenericAxisDataNew[HMI_AxisIndex].xActive				:= FALSE;
			HMI_MC_GenericAxisDataNew[HMI_AxisIndex].xBrakeReleased			:= FALSE;
			HMI_MC_GenericAxisDataNew[HMI_AxisIndex].xEnabled;
			HMI_MC_GenericAxisDataNew[HMI_AxisIndex].xFollowingError		:= FALSE;
			HMI_MC_GenericAxisDataNew[HMI_AxisIndex].xHomed					:= FALSE;
			HMI_MC_GenericAxisDataNew[HMI_AxisIndex].xInError				:= FALSE;
			HMI_MC_GenericAxisDataNew[HMI_AxisIndex].xInPosition			:= FALSE;
			HMI_MC_GenericAxisDataNew[HMI_AxisIndex].xPowered				:= FALSE;
			HMI_MC_GenericAxisDataNew[HMI_AxisIndex].xReal					:= FALSE;
			HMI_MC_GenericAxisDataNew[HMI_AxisIndex].xRunning				:= FALSE;
			HMI_MC_GenericAxisDataNew[HMI_AxisIndex].xSynchro				:= FALSE;
			HMI_MC_GenericAxisDataNew[HMI_AxisIndex].xTorqueError			:= FALSE;
			//HMI_MC_GenericAxisDataNew[HMI_AxisIndex].xHmiWait				:= TRUE;
			END_IF

			xAxisInVelocityControl	:= VAR_Machine.stOutletModule.iq_astSubModuleAxis[HMI_MC_GenericAxisDataNew[HMI_AxisIndex].uiAxisID - CST_OutletSubModuleHmiStart].iq_stStatus.q_stMainAxisStatus.q_xVelocityControl;

		END_IF
	END_FOR

		IF VAR_Machine.stFillerModule.iq_stStatus.q_xInitDone AND  VAR_Machine.stInletModule.iq_stStatus.q_xInitDone AND VAR_Machine.stOutletModule.iq_stStatus.q_xInitDone THEN//v1.7.2
			HMI_MC_GenericAxisData.xHmiWait										:= FALSE ;//v1.7.2
		ELSE //v1.7.2
			HMI_MC_GenericAxisData.xHmiWait										:= TRUE;//v1.7.2
		END_IF//v1.7.2

		/////////////////////////////////////////////////
		HMI_MC_EncoderDiagnostic.Present 									:= CFG_MC.Generic.SyncroPar.ExternalEncoder;
		HMI_MC_EncoderDiagnostic.ModuleOK 									:= MC_InputOutput.Network.Machine.Commands.MasterEncoderPositionValid;
		HMI_MC_EncoderDiagnostic.Value 										:= ITC_Motion_ExtEnc;

		HMI_MC_GenericAxisData.rPosition									:= LREAL_TO_REAL(VAR_Machine.stFillerModule.iq_astSubModuleAxis[15].iq_stStatus.q_stMainAxisStatus.q_lrPosition);//V4.A.A.1.7.0
	END_ACTION

(* ---- Init.st ---- *)
PROGRAM _INIT
	//Init of data struct

	HMI_MC_MachineStatus;
	HMI_MC_GenericAxisData;
	HMI_MC_AlarmList;

	HMI_MC_MachineStatus.rMachineStep	:=	LREAL_TO_REAL(CFG_MC.Mechanical.MachineStep);
END_PROGRAM

(* ---- Itc_Filler.st ---- *)
ACTION FillerInput:
	(* Commands *)
	VAR_Machine.stFillerModule.iq_stCmd.i_xFillerAbsolutePositionSensor		:= MC_InputOutput.Network.Filler.Commands.FillerAbsolutePositionSensor; (*//V4.A.A.1.6.12e*)
	VAR_Machine.stFillerModule.iq_stCmd.i_xRinserFillerAbsolutePosSensor	:= MC_InputOutput.Network.Filler.Commands.RinserAbsolutePositionSensor; (*//V4.A.A.1.6.12e*)
	VAR_Machine.stFillerModule.iq_stCmd.i_xCapperAbsolutePositionSensor		:= MC_InputOutput.Network.Filler.Commands.CapperAbsolutePositionSensor; (*//V4.A.A.1.6.12e*)
	VAR_Machine.stFillerModule.iq_stCmd.i_xCrownerAbsolutePositionSensor	:= MC_InputOutput.Network.Filler.Commands.CrownerAbsolutePositionSensor; (*//V4.A.A.1.6.12e*)
	VAR_Machine.stFillerModule.iq_stCmd.i_xDoserAbsolutePositionSensor		:= MC_InputOutput.Network.Filler.Commands.DoserAbsolutePositionSensor; (*//V4.A.A.1.6.12e*)

	VAR_Machine.stFillerModule.iq_stCmd.i_xVelocityAxisStop				:= MC_InputOutput.Network.Filler.Commands.VelocityAxisStop;

	FOR uiAxisIndex := CST_FirstFillerModuleAxis TO CST_LastFillerModuleAxis DO
		VAR_Machine.stFillerModule.iq_astSubModuleAxis[uiAxisIndex].iq_stStatus.q_stMainAxisStatus.iq_xNotErrEncoder	:= MC_InputOutput.Safety.Filler.Commands.AxesDiag[uiAxisIndex].DI_NotErrENC;
		VAR_Machine.stFillerModule.iq_astSubModuleAxis[uiAxisIndex].iq_stStatus.q_stMainAxisStatus.iq_xOperational		:= MC_InputOutput.Safety.Filler.Commands.AxesDiag[uiAxisIndex].DI_Operational;
		(* Parameters *)
		IF uiAxisIndex >= 15 THEN
			VAR_Machine.stFillerModule.iq_astSubModuleAxis[uiAxisIndex].iq_stParam.i_rVelocityOffsetFactor		:= MC_InputOutput.Network.Filler.Parameters.OutletConveyorKs / 100.0;
		ELSE
			VAR_Machine.stFillerModule.iq_astSubModuleAxis[uiAxisIndex].iq_stParam.i_rVelocityOffsetFactor		:= MC_InputOutput.Network.Filler.Parameters.InletConveyorKs / 100.0;
		END_IF
	END_FOR

	VAR_Machine.stFillerModule.iq_stParameters.i_uiFillerAbsolutePositionOffset	:= MC_InputOutput.Network.Filler.Parameters.FillerAbsolutePositionOffset; (*//V4.A.A.1.6.12e*)
	VAR_Machine.stFillerModule.iq_stParameters.i_uiFillerStepsNumber			:= MC_InputOutput.Network.Filler.Parameters.FillerStepsNumber; (*//V4.A.A.1.6.12e*)
	VAR_Machine.stFillerModule.iq_stParameters.i_uiRinserAbsolutePositionOffset	:= MC_InputOutput.Network.Filler.Parameters.RinserAbsolutePositionOffset; (*//V4.A.A.1.6.12e*)
	VAR_Machine.stFillerModule.iq_stParameters.i_uiRinserStepsNumber			:= MC_InputOutput.Network.Filler.Parameters.RinserStepsNumber; (*//V4.A.A.1.6.12e*)
	VAR_Machine.stFillerModule.iq_stParameters.i_uiCapperAbsolutePositionOffset	:= MC_InputOutput.Network.Filler.Parameters.CapperAbsolutePositionOffset; (*//V4.A.A.1.6.12e*)
	VAR_Machine.stFillerModule.iq_stParameters.i_uiCapperStepsNumber			:= MC_InputOutput.Network.Filler.Parameters.CapperStepsNumber; (*//V4.A.A.1.6.12e*)
	VAR_Machine.stFillerModule.iq_stParameters.i_uiCrownerAbsolutePosOffset		:= MC_InputOutput.Network.Filler.Parameters.CrownerAbsolutePositionOffset; (*//V4.A.A.1.6.12e*)
	VAR_Machine.stFillerModule.iq_stParameters.i_uiCrownerStepsNumber			:= MC_InputOutput.Network.Filler.Parameters.CrownerStepsNumber; (*//V4.A.A.1.6.12e*)
	VAR_Machine.stFillerModule.iq_stParameters.i_uiDoserPositionOffset			:= MC_InputOutput.Network.Filler.Parameters.DoserAbsolutePositionOffset; (*//V4.A.A.1.6.12e*)
	VAR_Machine.stFillerModule.iq_stParameters.i_uiDoserStepsNumber				:= MC_InputOutput.Network.Filler.Parameters.DoserStepsNumber; (*//V4.A.A.1.6.12e*)

	(*Disable axis Rinser command*)
	VAR_Machine.stFillerModule.iq_astSubModuleAxis[CFG_MC.Mechanical.ReferenceId.Rinser].iq_stCmd.i_xDisableAxis	:= MC_InputOutput.Network.Filler.Commands.DisableRinserAxis;//V4.A.A.1.7.0
	(*Disable axis Doser command*)
	VAR_Machine.stFillerModule.iq_astSubModuleAxis[CFG_MC.Mechanical.ReferenceId.Doser].iq_stCmd.i_xDisableAxis		:= MC_InputOutput.Network.Filler.Commands.DisableDoserAxis;//V4.A.A.1.7.0
	(*Disable axis Filler command*)
	VAR_Machine.stFillerModule.iq_astSubModuleAxis[CFG_MC.Mechanical.ReferenceId.Filler].iq_stCmd.i_xDisableAxis		:= MC_InputOutput.Network.Filler.Commands.DisableFillerAxis;//V4.A.A.1.7.0

	VAR_Machine.stFillerModule.iq_astSubModuleAxis[CST_MainAxis].iq_stParam.i_rTorqueErrorThreshold	:= MC_InputOutput.Network.Filler.Parameters.TorqueError.Main;
	FOR uiAxisIndex := 1 TO 10 DO
		VAR_Machine.stFillerModule.iq_astSubModuleAxis[(uiAxisIndex - 1) +  CST_FirstFillerModuleAxis].iq_stParam.i_rTorqueErrorThreshold	:= MC_InputOutput.Network.Filler.Parameters.TorqueError.In[uiAxisIndex];
	END_FOR

	FOR uiAxisIndex := 1 TO 6 DO
		VAR_Machine.stFillerModule.iq_astSubModuleAxis[(uiAxisIndex) + CST_MainAxis].iq_stParam.i_rTorqueErrorThreshold	:= MC_InputOutput.Network.Filler.Parameters.TorqueError.Out[uiAxisIndex];
	END_FOR
END_ACTION

ACTION FillerOutput:
	(* Filler status *)
	MC_InputOutput.Network.Filler.Status.Velocity						:= VAR_Machine.stFillerModule.iq_stStatus.q_rVelocity * 10.0;
	MC_InputOutput.Network.Filler.Status.FillerAbsolutePosition			:= VAR_Machine.stFillerModule.iq_stStatus.q_lrFillerAbsolutePosition; (*//V4.A.A.1.6.12e*)
	MC_InputOutput.Network.Filler.Status.RinserAbsolutePosition			:= VAR_Machine.stFillerModule.iq_stStatus.q_lrRinserAbsolutePosition; (*//V4.A.A.1.6.12e*)
	MC_InputOutput.Network.Filler.Status.CapperAbsolutePosition			:= VAR_Machine.stFillerModule.iq_stStatus.q_lrCapperAbsolutePosition; (*//V4.A.A.1.6.12e*)
	MC_InputOutput.Network.Filler.Status.CrownerAbsolutePosition		:= VAR_Machine.stFillerModule.iq_stStatus.q_lrCrownerAbsolutePosition; (*//V4.A.A.1.6.12e*)
	MC_InputOutput.Network.Filler.Status.DoserAbsolutePosition			:= VAR_Machine.stFillerModule.iq_stStatus.q_lrDoserAbsolutePosition; (*//V4.A.A.1.6.12e*)

	MC_InputOutput.Network.Filler.Status.ModuleHomed					:= VAR_Machine.stFillerModule.iq_stStatus.q_xModuleHomed;
	MC_InputOutput.Network.Filler.Status.ModuleInPosition;
	MC_InputOutput.Network.Filler.Status.ModulePowered					:= VAR_Machine.stFillerModule.iq_stStatus.q_xModulePowered;
	MC_InputOutput.Network.Filler.Status.ModuleReal						:= VAR_Machine.stFillerModule.iq_stStatus.q_xModuleReal;
	MC_InputOutput.Network.Filler.Status.ModuleRunning					:= SEL(VAR_Machine.iq_stStatus.q_xMultiModalityActive, VAR_Machine.iq_stStatus.q_xMachineStartFbk, VAR_Machine.stFillerModule.iq_stStatus.q_xModuleStartFbk);
	MC_InputOutput.Network.Filler.Status.ModuleNotInitialized			:= NOT VAR_Machine.stFillerModule.iq_stStatus.q_xInitDone;

	MC_InputOutput.Network.Filler.Status.AutoActive						:= VAR_Machine.stFillerModule.iq_stStatus.q_xAutoMultiActive;
	MC_InputOutput.Network.Filler.Status.ModuleJogActive				:= VAR_Machine.stFillerModule.iq_stStatus.q_xJogMultiActive;
	MC_InputOutput.Network.Filler.Status.SlowMotionActive				:= VAR_Machine.stFillerModule.iq_stStatus.q_xSlowMotionActive;

	MC_InputOutput.Network.Filler.Status.AutoCmdFeedback				:= VAR_Machine.stFillerModule.iq_stStatus.q_xAutoMultiActive AND VAR_Machine.stFillerModule.iq_stCmd.i_xStart;
	MC_InputOutput.Network.Filler.Status.JogCmdFeedback					:= VAR_Machine.stFillerModule.iq_stStatus.q_xJogMultiActive AND VAR_Machine.stFillerModule.iq_stCmd.i_xJogPB;

	MC_InputOutput.Network.Filler.Status.CarouselReal					:= VAR_Machine.stFillerModule.iq_astSubModuleAxis[CST_MainAxis].iq_stStatus.q_stMainAxisStatus.q_xAxisReal;
	MC_InputOutput.Network.Filler.Status.In01Real					:= VAR_Machine.stFillerModule.iq_astSubModuleAxis[CST_Inlet01].iq_stStatus.q_stMainAxisStatus.q_xAxisReal;
	MC_InputOutput.Network.Filler.Status.In02Real					:= VAR_Machine.stFillerModule.iq_astSubModuleAxis[CST_Inlet02].iq_stStatus.q_stMainAxisStatus.q_xAxisReal;
	MC_InputOutput.Network.Filler.Status.In03Real					:= VAR_Machine.stFillerModule.iq_astSubModuleAxis[CST_Inlet03].iq_stStatus.q_stMainAxisStatus.q_xAxisReal;
	MC_InputOutput.Network.Filler.Status.In04Real					:= VAR_Machine.stFillerModule.iq_astSubModuleAxis[CST_Inlet04].iq_stStatus.q_stMainAxisStatus.q_xAxisReal;
	MC_InputOutput.Network.Filler.Status.In05Real					:= VAR_Machine.stFillerModule.iq_astSubModuleAxis[CST_Inlet05].iq_stStatus.q_stMainAxisStatus.q_xAxisReal;
	MC_InputOutput.Network.Filler.Status.In06Real					:= VAR_Machine.stFillerModule.iq_astSubModuleAxis[CST_Inlet06].iq_stStatus.q_stMainAxisStatus.q_xAxisReal;
	MC_InputOutput.Network.Filler.Status.In07Real					:= VAR_Machine.stFillerModule.iq_astSubModuleAxis[CST_Inlet07].iq_stStatus.q_stMainAxisStatus.q_xAxisReal;
	MC_InputOutput.Network.Filler.Status.In08Real					:= VAR_Machine.stFillerModule.iq_astSubModuleAxis[CST_Inlet08].iq_stStatus.q_stMainAxisStatus.q_xAxisReal;
	MC_InputOutput.Network.Filler.Status.In09Real					:= VAR_Machine.stFillerModule.iq_astSubModuleAxis[CST_Inlet09].iq_stStatus.q_stMainAxisStatus.q_xAxisReal;
	MC_InputOutput.Network.Filler.Status.In10Real					:= VAR_Machine.stFillerModule.iq_astSubModuleAxis[CST_Inlet10].iq_stStatus.q_stMainAxisStatus.q_xAxisReal;
	MC_InputOutput.Network.Filler.Status.Out01Real					:= VAR_Machine.stFillerModule.iq_astSubModuleAxis[CST_Outlet01].iq_stStatus.q_stMainAxisStatus.q_xAxisReal;
	MC_InputOutput.Network.Filler.Status.Out02Real					:= VAR_Machine.stFillerModule.iq_astSubModuleAxis[CST_Outlet02].iq_stStatus.q_stMainAxisStatus.q_xAxisReal;
	MC_InputOutput.Network.Filler.Status.Out03Real					:= VAR_Machine.stFillerModule.iq_astSubModuleAxis[CST_Outlet03].iq_stStatus.q_stMainAxisStatus.q_xAxisReal;
	MC_InputOutput.Network.Filler.Status.Out04Real					:= VAR_Machine.stFillerModule.iq_astSubModuleAxis[CST_Outlet04].iq_stStatus.q_stMainAxisStatus.q_xAxisReal;
	MC_InputOutput.Network.Filler.Status.Out05Real					:= VAR_Machine.stFillerModule.iq_astSubModuleAxis[CST_Outlet05].iq_stStatus.q_stMainAxisStatus.q_xAxisReal;
	MC_InputOutput.Network.Filler.Status.Out06Real					:= VAR_Machine.stFillerModule.iq_astSubModuleAxis[CST_Outlet06].iq_stStatus.q_stMainAxisStatus.q_xAxisReal;

	MC_InputOutput.Network.Filler.Status.FillerAbsolutePositionValid			:= VAR_Machine.stFillerModule.iq_stStatus.q_xFillerAbsolutePositionValid; (*//V4.A.A.1.6.12e*)
	MC_InputOutput.Network.Filler.Status.RinserAbsolutePositionValid			:= VAR_Machine.stFillerModule.iq_stStatus.q_xRinserAbsolutePositionValid; (*//V4.A.A.1.6.12e*)
	MC_InputOutput.Network.Filler.Status.CapperAbsolutePositionValid			:= VAR_Machine.stFillerModule.iq_stStatus.q_xCapperAbsolutePositionValid; (*//V4.A.A.1.6.12e*)
	MC_InputOutput.Network.Filler.Status.CrownerAbsolutePositionValid			:= VAR_Machine.stFillerModule.iq_stStatus.q_xCrownerAbsolutePositionValid; (*//V4.A.A.1.6.12e*)
	MC_InputOutput.Network.Filler.Status.DoserAbsolutePositionValid				:= VAR_Machine.stFillerModule.iq_stStatus.q_xDoserAbsolutePositionValid; (*//V4.A.A.1.6.12e*)

	(* Disabel Axis FeedBack *) //V4.A.A.1.7.0 Motion

	MC_InputOutput.Network.Filler.Status.RinserAxisDisabled						:= VAR_Machine.stFillerModule.iq_astSubModuleAxis[CFG_MC.Mechanical.ReferenceId.Rinser].iq_stStatus.q_stMainAxisStatus.q_xAxisDisabled;

	MC_InputOutput.Network.Filler.Status.DoserAxisDisabled						:= VAR_Machine.stFillerModule.iq_astSubModuleAxis[CFG_MC.Mechanical.ReferenceId.Doser].iq_stStatus.q_stMainAxisStatus.q_xAxisDisabled;
	MC_InputOutput.Network.Filler.Status.FillerAxisDisabled						:= VAR_Machine.stFillerModule.iq_astSubModuleAxis[CFG_MC.Mechanical.ReferenceId.Filler].iq_stStatus.q_stMainAxisStatus.q_xAxisDisabled;

	(* Button Enable *)
	MC_InputOutput.Network.Filler.Status.EnableAutoModality				:= NOT VAR_Machine.stFillerModule.iq_stStatus.q_xReactionActive;
	MC_InputOutput.Network.Filler.Status.EnableJogModality				:= VAR_Machine.stFillerModule.iq_stStatus.q_xModuleStopped AND
																			NOT VAR_Machine.stFillerModule.iq_stStatus.q_xReactionActive;

	(* Exception *)
	(* Main axis exception *)
	MC_InputOutput.Network.Filler.Exceptions.CarouselNotInOpException			:= NOT VAR_Machine.stFillerModule.iq_astSubModuleAxis[CST_MainAxis].iq_stStatus.q_stMainAxisStatus.iq_xOperational;
	MC_InputOutput.Network.Filler.Exceptions.CarouselSafetyException			:= NOT MC_InputOutput.Safety.Filler.Commands.AxesDiag[CST_MainAxis].DI_NotErrFUNC;
	MC_InputOutput.Network.Filler.Exceptions.CarouselTorqueException			:= VAR_Machine.stFillerModule.iq_astSubModuleAxis[CST_MainAxis].iq_stStatus.q_stMainAxisStatus.q_xTorqueError;
	MC_InputOutput.Network.Filler.Exceptions.CarouselTrackException				:= VAR_Machine.stFillerModule.iq_astSubModuleAxis[CST_MainAxis].iq_stStatus.q_stMainAxisStatus.q_xLagError;
	MC_InputOutput.Network.Filler.Exceptions.CarouselDriveException				:= VAR_Machine.stFillerModule.iq_astSubModuleAxis[CST_MainAxis].iq_stStatus.q_stMainAxisStatus.q_xError;
	MC_InputOutput.Network.Filler.Exceptions.CarouselHomeException				:= NOT VAR_Machine.stFillerModule.iq_astSubModuleAxis[CST_MainAxis].iq_stStatus.q_stMainAxisStatus.q_xIsHomed AND
																					VAR_Machine.stFillerModule.iq_astSubModuleAxis[CST_MainAxis].iq_stStatus.q_stMainAxisStatus.q_xInitDone;

	(* Inlet axis exception *)
	IF VAR_Machine.stFillerModule.iq_astSubModuleAxis[CST_Inlet01].iq_stStatus.q_stMainAxisStatus.q_xAxisReal THEN
		IF NOT CFG_MC.Axes.Filler.In[1].VelocityControl THEN
			MC_InputOutput.Network.Filler.Exceptions.Inlet01NotInOpException			:= NOT VAR_Machine.stFillerModule.iq_astSubModuleAxis[CST_Inlet01].iq_stStatus.q_stMainAxisStatus.iq_xOperational;
			MC_InputOutput.Network.Filler.Exceptions.Inlet01SafetyException				:= NOT MC_InputOutput.Safety.Filler.Commands.AxesDiag[CST_Inlet01].DI_NotErrFUNC;
		END_IF
		MC_InputOutput.Network.Filler.Exceptions.Inlet01TorqueException				:= VAR_Machine.stFillerModule.iq_astSubModuleAxis[CST_Inlet01].iq_stStatus.q_stMainAxisStatus.q_xTorqueError;
		MC_InputOutput.Network.Filler.Exceptions.Inlet01TrackException				:= VAR_Machine.stFillerModule.iq_astSubModuleAxis[CST_Inlet01].iq_stStatus.q_stMainAxisStatus.q_xLagError;
		MC_InputOutput.Network.Filler.Exceptions.Inlet01DriveException				:= VAR_Machine.stFillerModule.iq_astSubModuleAxis[CST_Inlet01].iq_stStatus.q_stMainAxisStatus.q_xError;
		MC_InputOutput.Network.Filler.Exceptions.Inlet01HomeException				:= NOT VAR_Machine.stFillerModule.iq_astSubModuleAxis[CST_Inlet01].iq_stStatus.q_stMainAxisStatus.q_xIsHomed AND
																						VAR_Machine.stFillerModule.iq_astSubModuleAxis[CST_Inlet01].iq_stStatus.q_stMainAxisStatus.q_xInitDone;
	END_IF

	IF VAR_Machine.stFillerModule.iq_astSubModuleAxis[CST_Inlet02].iq_stStatus.q_stMainAxisStatus.q_xAxisReal THEN
		IF NOT CFG_MC.Axes.Filler.In[2].VelocityControl THEN
			MC_InputOutput.Network.Filler.Exceptions.Inlet02NotInOpException			:= NOT VAR_Machine.stFillerModule.iq_astSubModuleAxis[CST_Inlet02].iq_stStatus.q_stMainAxisStatus.iq_xOperational;
			MC_InputOutput.Network.Filler.Exceptions.Inlet02SafetyException				:= NOT MC_InputOutput.Safety.Filler.Commands.AxesDiag[CST_Inlet02].DI_NotErrFUNC;
		END_IF
		MC_InputOutput.Network.Filler.Exceptions.Inlet02TorqueException				:= VAR_Machine.stFillerModule.iq_astSubModuleAxis[CST_Inlet02].iq_stStatus.q_stMainAxisStatus.q_xTorqueError;
		MC_InputOutput.Network.Filler.Exceptions.Inlet02TrackException				:= VAR_Machine.stFillerModule.iq_astSubModuleAxis[CST_Inlet02].iq_stStatus.q_stMainAxisStatus.q_xLagError;
		MC_InputOutput.Network.Filler.Exceptions.Inlet02DriveException				:= VAR_Machine.stFillerModule.iq_astSubModuleAxis[CST_Inlet02].iq_stStatus.q_stMainAxisStatus.q_xError;
		MC_InputOutput.Network.Filler.Exceptions.Inlet02HomeException				:= NOT VAR_Machine.stFillerModule.iq_astSubModuleAxis[CST_Inlet02].iq_stStatus.q_stMainAxisStatus.q_xIsHomed AND
																						VAR_Machine.stFillerModule.iq_astSubModuleAxis[CST_Inlet02].iq_stStatus.q_stMainAxisStatus.q_xInitDone;
	END_IF

	IF VAR_Machine.stFillerModule.iq_astSubModuleAxis[CST_Inlet03].iq_stStatus.q_stMainAxisStatus.q_xAxisReal THEN
		IF NOT CFG_MC.Axes.Filler.In[3].VelocityControl THEN
			MC_InputOutput.Network.Filler.Exceptions.Inlet03NotInOpException			:= NOT VAR_Machine.stFillerModule.iq_astSubModuleAxis[CST_Inlet03].iq_stStatus.q_stMainAxisStatus.iq_xOperational;
			MC_InputOutput.Network.Filler.Exceptions.Inlet03SafetyException				:= NOT MC_InputOutput.Safety.Filler.Commands.AxesDiag[CST_Inlet03].DI_NotErrFUNC;
		END_IF
		MC_InputOutput.Network.Filler.Exceptions.Inlet03TorqueException				:= VAR_Machine.stFillerModule.iq_astSubModuleAxis[CST_Inlet03].iq_stStatus.q_stMainAxisStatus.q_xTorqueError;
		MC_InputOutput.Network.Filler.Exceptions.Inlet03TrackException				:= VAR_Machine.stFillerModule.iq_astSubModuleAxis[CST_Inlet03].iq_stStatus.q_stMainAxisStatus.q_xLagError;
		MC_InputOutput.Network.Filler.Exceptions.Inlet03DriveException				:= VAR_Machine.stFillerModule.iq_astSubModuleAxis[CST_Inlet03].iq_stStatus.q_stMainAxisStatus.q_xError;
		MC_InputOutput.Network.Filler.Exceptions.Inlet03HomeException				:= NOT VAR_Machine.stFillerModule.iq_astSubModuleAxis[CST_Inlet03].iq_stStatus.q_stMainAxisStatus.q_xIsHomed AND
																						VAR_Machine.stFillerModule.iq_astSubModuleAxis[CST_Inlet03].iq_stStatus.q_stMainAxisStatus.q_xInitDone;
	END_IF

	IF VAR_Machine.stFillerModule.iq_astSubModuleAxis[CST_Inlet04].iq_stStatus.q_stMainAxisStatus.q_xAxisReal THEN
		IF NOT CFG_MC.Axes.Filler.In[4].VelocityControl THEN
			MC_InputOutput.Network.Filler.Exceptions.Inlet04NotInOpException			:= NOT VAR_Machine.stFillerModule.iq_astSubModuleAxis[CST_Inlet04].iq_stStatus.q_stMainAxisStatus.iq_xOperational;
			MC_InputOutput.Network.Filler.Exceptions.Inlet04SafetyException				:= NOT MC_InputOutput.Safety.Filler.Commands.AxesDiag[CST_Inlet04].DI_NotErrFUNC;
		END_IF
		MC_InputOutput.Network.Filler.Exceptions.Inlet04DriveException				:= VAR_Machine.stFillerModule.iq_astSubModuleAxis[CST_Inlet04].iq_stStatus.q_stMainAxisStatus.q_xError;
		MC_InputOutput.Network.Filler.Exceptions.Inlet04TorqueException				:= VAR_Machine.stFillerModule.iq_astSubModuleAxis[CST_Inlet04].iq_stStatus.q_stMainAxisStatus.q_xTorqueError;
		MC_InputOutput.Network.Filler.Exceptions.Inlet04TrackException				:= VAR_Machine.stFillerModule.iq_astSubModuleAxis[CST_Inlet04].iq_stStatus.q_stMainAxisStatus.q_xLagError;
		MC_InputOutput.Network.Filler.Exceptions.Inlet04HomeException 				:= NOT VAR_Machine.stFillerModule.iq_astSubModuleAxis[CST_Inlet04].iq_stStatus.q_stMainAxisStatus.q_xIsHomed AND
																						VAR_Machine.stFillerModule.iq_astSubModuleAxis[CST_Inlet04].iq_stStatus.q_stMainAxisStatus.q_xInitDone;
	END_IF

	IF VAR_Machine.stFillerModule.iq_astSubModuleAxis[CST_Inlet05].iq_stStatus.q_stMainAxisStatus.q_xAxisReal THEN
		IF NOT CFG_MC.Axes.Filler.In[5].VelocityControl THEN
			MC_InputOutput.Network.Filler.Exceptions.Inlet05NotInOpException			:= NOT VAR_Machine.stFillerModule.iq_astSubModuleAxis[CST_Inlet05].iq_stStatus.q_stMainAxisStatus.iq_xOperational;
			MC_InputOutput.Network.Filler.Exceptions.Inlet05SafetyException				:= NOT MC_InputOutput.Safety.Filler.Commands.AxesDiag[CST_Inlet05].DI_NotErrFUNC;
		END_IF
	MC_InputOutput.Network.Filler.Exceptions.Inlet05DriveException				:= VAR_Machine.stFillerModule.iq_astSubModuleAxis[CST_Inlet05].iq_stStatus.q_stMainAxisStatus.q_xError;
	MC_InputOutput.Network.Filler.Exceptions.Inlet05TorqueException				:= VAR_Machine.stFillerModule.iq_astSubModuleAxis[CST_Inlet05].iq_stStatus.q_stMainAxisStatus.q_xTorqueError;
	MC_InputOutput.Network.Filler.Exceptions.Inlet05TrackException				:= VAR_Machine.stFillerModule.iq_astSubModuleAxis[CST_Inlet05].iq_stStatus.q_stMainAxisStatus.q_xLagError;
	MC_InputOutput.Network.Filler.Exceptions.Inlet05HomeException				:= NOT VAR_Machine.stFillerModule.iq_astSubModuleAxis[CST_Inlet05].iq_stStatus.q_stMainAxisStatus.q_xIsHomed AND
																					VAR_Machine.stFillerModule.iq_astSubModuleAxis[CST_Inlet05].iq_stStatus.q_stMainAxisStatus.q_xInitDone;
	END_IF

	IF VAR_Machine.stFillerModule.iq_astSubModuleAxis[CST_Inlet06].iq_stStatus.q_stMainAxisStatus.q_xAxisReal THEN
		IF NOT CFG_MC.Axes.Filler.In[6].VelocityControl THEN
			MC_InputOutput.Network.Filler.Exceptions.Inlet06NotInOpException			:= NOT VAR_Machine.stFillerModule.iq_astSubModuleAxis[CST_Inlet06].iq_stStatus.q_stMainAxisStatus.iq_xOperational;
			MC_InputOutput.Network.Filler.Exceptions.Inlet06SafetyException				:= NOT MC_InputOutput.Safety.Filler.Commands.AxesDiag[CST_Inlet06].DI_NotErrFUNC;
		END_IF
		MC_InputOutput.Network.Filler.Exceptions.Inlet06DriveException				:= VAR_Machine.stFillerModule.iq_astSubModuleAxis[CST_Inlet06].iq_stStatus.q_stMainAxisStatus.q_xError;
		MC_InputOutput.Network.Filler.Exceptions.Inlet06TorqueException				:= VAR_Machine.stFillerModule.iq_astSubModuleAxis[CST_Inlet06].iq_stStatus.q_stMainAxisStatus.q_xTorqueError;
		MC_InputOutput.Network.Filler.Exceptions.Inlet06TrackException				:= VAR_Machine.stFillerModule.iq_astSubModuleAxis[CST_Inlet06].iq_stStatus.q_stMainAxisStatus.q_xLagError;
		MC_InputOutput.Network.Filler.Exceptions.Inlet06HomeException				:= NOT VAR_Machine.stFillerModule.iq_astSubModuleAxis[CST_Inlet06].iq_stStatus.q_stMainAxisStatus.q_xIsHomed AND
																						VAR_Machine.stFillerModule.iq_astSubModuleAxis[CST_Inlet06].iq_stStatus.q_stMainAxisStatus.q_xInitDone;
	END_IF

	IF VAR_Machine.stFillerModule.iq_astSubModuleAxis[CST_Inlet07].iq_stStatus.q_stMainAxisStatus.q_xAxisReal THEN
		IF NOT CFG_MC.Axes.Filler.In[7].VelocityControl THEN
			MC_InputOutput.Network.Filler.Exceptions.Inlet07NotInOpException			:= NOT VAR_Machine.stFillerModule.iq_astSubModuleAxis[CST_Inlet07].iq_stStatus.q_stMainAxisStatus.iq_xOperational;
			MC_InputOutput.Network.Filler.Exceptions.Inlet07SafetyException				:= NOT MC_InputOutput.Safety.Filler.Commands.AxesDiag[CST_Inlet07].DI_NotErrFUNC;
		END_IF
		MC_InputOutput.Network.Filler.Exceptions.Inlet07DriveException				:= VAR_Machine.stFillerModule.iq_astSubModuleAxis[CST_Inlet07].iq_stStatus.q_stMainAxisStatus.q_xError;
		MC_InputOutput.Network.Filler.Exceptions.Inlet07TorqueException				:= VAR_Machine.stFillerModule.iq_astSubModuleAxis[CST_Inlet07].iq_stStatus.q_stMainAxisStatus.q_xTorqueError;
		MC_InputOutput.Network.Filler.Exceptions.Inlet07TrackException				:= VAR_Machine.stFillerModule.iq_astSubModuleAxis[CST_Inlet07].iq_stStatus.q_stMainAxisStatus.q_xLagError;
		MC_InputOutput.Network.Filler.Exceptions.Inlet07HomeException				:= NOT VAR_Machine.stFillerModule.iq_astSubModuleAxis[CST_Inlet07].iq_stStatus.q_stMainAxisStatus.q_xIsHomed AND
																						VAR_Machine.stFillerModule.iq_astSubModuleAxis[CST_Inlet07].iq_stStatus.q_stMainAxisStatus.q_xInitDone;
	END_IF

	IF VAR_Machine.stFillerModule.iq_astSubModuleAxis[CST_Inlet08].iq_stStatus.q_stMainAxisStatus.q_xAxisReal THEN
		IF NOT CFG_MC.Axes.Filler.In[8].VelocityControl THEN
			MC_InputOutput.Network.Filler.Exceptions.Inlet08NotInOpException			:= NOT VAR_Machine.stFillerModule.iq_astSubModuleAxis[CST_Inlet08].iq_stStatus.q_stMainAxisStatus.iq_xOperational;
			MC_InputOutput.Network.Filler.Exceptions.Inlet08SafetyException				:= NOT MC_InputOutput.Safety.Filler.Commands.AxesDiag[CST_Inlet08].DI_NotErrFUNC;
		END_IF
		MC_InputOutput.Network.Filler.Exceptions.Inlet08DriveException				:= VAR_Machine.stFillerModule.iq_astSubModuleAxis[CST_Inlet08].iq_stStatus.q_stMainAxisStatus.q_xError;
		MC_InputOutput.Network.Filler.Exceptions.Inlet08TorqueException				:= VAR_Machine.stFillerModule.iq_astSubModuleAxis[CST_Inlet08].iq_stStatus.q_stMainAxisStatus.q_xTorqueError;
		MC_InputOutput.Network.Filler.Exceptions.Inlet08TrackException				:= VAR_Machine.stFillerModule.iq_astSubModuleAxis[CST_Inlet08].iq_stStatus.q_stMainAxisStatus.q_xLagError;
		MC_InputOutput.Network.Filler.Exceptions.Inlet08HomeException				:= NOT VAR_Machine.stFillerModule.iq_astSubModuleAxis[CST_Inlet08].iq_stStatus.q_stMainAxisStatus.q_xIsHomed AND
																						VAR_Machine.stFillerModule.iq_astSubModuleAxis[CST_Inlet08].iq_stStatus.q_stMainAxisStatus.q_xInitDone;
	END_IF

	IF VAR_Machine.stFillerModule.iq_astSubModuleAxis[CST_Inlet09].iq_stStatus.q_stMainAxisStatus.q_xAxisReal THEN
		IF NOT CFG_MC.Axes.Filler.In[9].VelocityControl THEN
			MC_InputOutput.Network.Filler.Exceptions.Inlet09NotInOpException			:= NOT VAR_Machine.stFillerModule.iq_astSubModuleAxis[CST_Inlet09].iq_stStatus.q_stMainAxisStatus.iq_xOperational;
			MC_InputOutput.Network.Filler.Exceptions.Inlet09SafetyException				:= NOT MC_InputOutput.Safety.Filler.Commands.AxesDiag[CST_Inlet09].DI_NotErrFUNC;
		END_IF
		MC_InputOutput.Network.Filler.Exceptions.Inlet09DriveException				:= VAR_Machine.stFillerModule.iq_astSubModuleAxis[CST_Inlet09].iq_stStatus.q_stMainAxisStatus.q_xError;
		MC_InputOutput.Network.Filler.Exceptions.Inlet09TorqueException				:= VAR_Machine.stFillerModule.iq_astSubModuleAxis[CST_Inlet09].iq_stStatus.q_stMainAxisStatus.q_xTorqueError;
		MC_InputOutput.Network.Filler.Exceptions.Inlet09TrackException				:= VAR_Machine.stFillerModule.iq_astSubModuleAxis[CST_Inlet09].iq_stStatus.q_stMainAxisStatus.q_xLagError;
		MC_InputOutput.Network.Filler.Exceptions.Inlet09HomeException				:= NOT VAR_Machine.stFillerModule.iq_astSubModuleAxis[CST_Inlet09].iq_stStatus.q_stMainAxisStatus.q_xIsHomed AND
																					VAR_Machine.stFillerModule.iq_astSubModuleAxis[CST_Inlet09].iq_stStatus.q_stMainAxisStatus.q_xInitDone;
	END_IF

	IF VAR_Machine.stFillerModule.iq_astSubModuleAxis[CST_Inlet10].iq_stStatus.q_stMainAxisStatus.q_xAxisReal THEN
		IF NOT CFG_MC.Axes.Filler.In[10].VelocityControl THEN
			MC_InputOutput.Network.Filler.Exceptions.Inlet10NotInOpException			:= NOT VAR_Machine.stFillerModule.iq_astSubModuleAxis[CST_Inlet10].iq_stStatus.q_stMainAxisStatus.iq_xOperational;
			MC_InputOutput.Network.Filler.Exceptions.Inlet10SafetyException				:= NOT MC_InputOutput.Safety.Filler.Commands.AxesDiag[CST_Inlet10].DI_NotErrFUNC;
		END_IF
		MC_InputOutput.Network.Filler.Exceptions.Inlet10DriveException				:= VAR_Machine.stFillerModule.iq_astSubModuleAxis[CST_Inlet10].iq_stStatus.q_stMainAxisStatus.q_xError;
		MC_InputOutput.Network.Filler.Exceptions.Inlet10TorqueException				:= VAR_Machine.stFillerModule.iq_astSubModuleAxis[CST_Inlet10].iq_stStatus.q_stMainAxisStatus.q_xTorqueError;
		MC_InputOutput.Network.Filler.Exceptions.Inlet10TrackException				:= VAR_Machine.stFillerModule.iq_astSubModuleAxis[CST_Inlet10].iq_stStatus.q_stMainAxisStatus.q_xLagError;
		MC_InputOutput.Network.Filler.Exceptions.Inlet10HomeException				:= NOT VAR_Machine.stFillerModule.iq_astSubModuleAxis[CST_Inlet10].iq_stStatus.q_stMainAxisStatus.q_xIsHomed AND
																						VAR_Machine.stFillerModule.iq_astSubModuleAxis[CST_Inlet10].iq_stStatus.q_stMainAxisStatus.q_xInitDone;
	END_IF

	(* Outlet axis exception *)
	IF VAR_Machine.stFillerModule.iq_astSubModuleAxis[CST_Outlet01].iq_stStatus.q_stMainAxisStatus.q_xAxisReal THEN
		IF NOT CFG_MC.Axes.Filler.Out[1].VelocityControl THEN
			MC_InputOutput.Network.Filler.Exceptions.Outlet01NotInOpException			:= NOT VAR_Machine.stFillerModule.iq_astSubModuleAxis[CST_Outlet01].iq_stStatus.q_stMainAxisStatus.iq_xOperational;
			MC_InputOutput.Network.Filler.Exceptions.Outlet01SafetyException			:= NOT MC_InputOutput.Safety.Filler.Commands.AxesDiag[CST_Outlet01].DI_NotErrFUNC;
		END_IF
		MC_InputOutput.Network.Filler.Exceptions.Outlet01DriveException				:= VAR_Machine.stFillerModule.iq_astSubModuleAxis[CST_Outlet01].iq_stStatus.q_stMainAxisStatus.q_xError;
		MC_InputOutput.Network.Filler.Exceptions.Outlet01TorqueException			:= VAR_Machine.stFillerModule.iq_astSubModuleAxis[CST_Outlet01].iq_stStatus.q_stMainAxisStatus.q_xTorqueError;
		MC_InputOutput.Network.Filler.Exceptions.Outlet01TrackException				:= VAR_Machine.stFillerModule.iq_astSubModuleAxis[CST_Outlet01].iq_stStatus.q_stMainAxisStatus.q_xLagError;
		MC_InputOutput.Network.Filler.Exceptions.Outlet01HomeException				:= NOT VAR_Machine.stFillerModule.iq_astSubModuleAxis[CST_Outlet01].iq_stStatus.q_stMainAxisStatus.q_xIsHomed AND
																						VAR_Machine.stFillerModule.iq_astSubModuleAxis[CST_Outlet01].iq_stStatus.q_stMainAxisStatus.q_xInitDone;
	END_IF

	IF VAR_Machine.stFillerModule.iq_astSubModuleAxis[CST_Outlet02].iq_stStatus.q_stMainAxisStatus.q_xAxisReal THEN
		IF NOT CFG_MC.Axes.Filler.Out[2].VelocityControl THEN
			MC_InputOutput.Network.Filler.Exceptions.Outlet02NotInOpException			:= NOT VAR_Machine.stFillerModule.iq_astSubModuleAxis[CST_Outlet02].iq_stStatus.q_stMainAxisStatus.iq_xOperational;
			MC_InputOutput.Network.Filler.Exceptions.Outlet02SafetyException			:= NOT MC_InputOutput.Safety.Filler.Commands.AxesDiag[CST_Outlet02].DI_NotErrFUNC;
		END_IF
		MC_InputOutput.Network.Filler.Exceptions.Outlet02DriveException 			:= VAR_Machine.stFillerModule.iq_astSubModuleAxis[CST_Outlet02].iq_stStatus.q_stMainAxisStatus.q_xError;
		MC_InputOutput.Network.Filler.Exceptions.Outlet02TorqueException			:= VAR_Machine.stFillerModule.iq_astSubModuleAxis[CST_Outlet02].iq_stStatus.q_stMainAxisStatus.q_xTorqueError;
		MC_InputOutput.Network.Filler.Exceptions.Outlet02TrackException 			:= VAR_Machine.stFillerModule.iq_astSubModuleAxis[CST_Outlet02].iq_stStatus.q_stMainAxisStatus.q_xLagError;
		MC_InputOutput.Network.Filler.Exceptions.Outlet02HomeException				:= NOT VAR_Machine.stFillerModule.iq_astSubModuleAxis[CST_Outlet02].iq_stStatus.q_stMainAxisStatus.q_xIsHomed AND
																						VAR_Machine.stFillerModule.iq_astSubModuleAxis[CST_Outlet02].iq_stStatus.q_stMainAxisStatus.q_xInitDone;
	END_IF

	IF VAR_Machine.stFillerModule.iq_astSubModuleAxis[CST_Outlet03].iq_stStatus.q_stMainAxisStatus.q_xAxisReal THEN
		IF NOT CFG_MC.Axes.Filler.Out[3].VelocityControl THEN
			MC_InputOutput.Network.Filler.Exceptions.Outlet03NotInOpException			:= NOT VAR_Machine.stFillerModule.iq_astSubModuleAxis[CST_Outlet03].iq_stStatus.q_stMainAxisStatus.iq_xOperational;
			MC_InputOutput.Network.Filler.Exceptions.Outlet03SafetyException			:= NOT MC_InputOutput.Safety.Filler.Commands.AxesDiag[CST_Outlet03].DI_NotErrFUNC;
		END_IF
		MC_InputOutput.Network.Filler.Exceptions.Outlet03DriveException				:= VAR_Machine.stFillerModule.iq_astSubModuleAxis[CST_Outlet03].iq_stStatus.q_stMainAxisStatus.q_xError;
		MC_InputOutput.Network.Filler.Exceptions.Outlet03TorqueException			:= VAR_Machine.stFillerModule.iq_astSubModuleAxis[CST_Outlet03].iq_stStatus.q_stMainAxisStatus.q_xTorqueError;
		MC_InputOutput.Network.Filler.Exceptions.Outlet03TrackException				:= VAR_Machine.stFillerModule.iq_astSubModuleAxis[CST_Outlet03].iq_stStatus.q_stMainAxisStatus.q_xLagError;
		MC_InputOutput.Network.Filler.Exceptions.Outlet03HomeException				:= NOT VAR_Machine.stFillerModule.iq_astSubModuleAxis[CST_Outlet03].iq_stStatus.q_stMainAxisStatus.q_xIsHomed AND
																						VAR_Machine.stFillerModule.iq_astSubModuleAxis[CST_Outlet03].iq_stStatus.q_stMainAxisStatus.q_xInitDone;
	END_IF

	IF VAR_Machine.stFillerModule.iq_astSubModuleAxis[CST_Outlet04].iq_stStatus.q_stMainAxisStatus.q_xAxisReal THEN
		IF NOT CFG_MC.Axes.Filler.Out[4].VelocityControl THEN
			MC_InputOutput.Network.Filler.Exceptions.Outlet04NotInOpException			:= NOT VAR_Machine.stFillerModule.iq_astSubModuleAxis[CST_Outlet04].iq_stStatus.q_stMainAxisStatus.iq_xOperational;
			MC_InputOutput.Network.Filler.Exceptions.Outlet04SafetyException			:= NOT MC_InputOutput.Safety.Filler.Commands.AxesDiag[CST_Outlet04].DI_NotErrFUNC;
		END_IF
		MC_InputOutput.Network.Filler.Exceptions.Outlet04DriveException 			:= VAR_Machine.stFillerModule.iq_astSubModuleAxis[CST_Outlet04].iq_stStatus.q_stMainAxisStatus.q_xError;
		MC_InputOutput.Network.Filler.Exceptions.Outlet04TorqueException			:= VAR_Machine.stFillerModule.iq_astSubModuleAxis[CST_Outlet04].iq_stStatus.q_stMainAxisStatus.q_xTorqueError;
		MC_InputOutput.Network.Filler.Exceptions.Outlet04TrackException 			:= VAR_Machine.stFillerModule.iq_astSubModuleAxis[CST_Outlet04].iq_stStatus.q_stMainAxisStatus.q_xLagError;
		MC_InputOutput.Network.Filler.Exceptions.Outlet04HomeException				:= NOT VAR_Machine.stFillerModule.iq_astSubModuleAxis[CST_Outlet04].iq_stStatus.q_stMainAxisStatus.q_xIsHomed AND
																						VAR_Machine.stFillerModule.iq_astSubModuleAxis[CST_Outlet04].iq_stStatus.q_stMainAxisStatus.q_xInitDone;
	END_IF

	IF VAR_Machine.stFillerModule.iq_astSubModuleAxis[CST_Outlet05].iq_stStatus.q_stMainAxisStatus.q_xAxisReal THEN
		IF NOT CFG_MC.Axes.Filler.Out[5].VelocityControl THEN
			MC_InputOutput.Network.Filler.Exceptions.Outlet05NotInOpException			:= NOT VAR_Machine.stFillerModule.iq_astSubModuleAxis[CST_Outlet05].iq_stStatus.q_stMainAxisStatus.iq_xOperational;
			MC_InputOutput.Network.Filler.Exceptions.Outlet05SafetyException			:= NOT MC_InputOutput.Safety.Filler.Commands.AxesDiag[CST_Outlet05].DI_NotErrFUNC;
		END_IF
		MC_InputOutput.Network.Filler.Exceptions.Outlet05DriveException				:= VAR_Machine.stFillerModule.iq_astSubModuleAxis[CST_Outlet05].iq_stStatus.q_stMainAxisStatus.q_xError;
		MC_InputOutput.Network.Filler.Exceptions.Outlet05TorqueException			:= VAR_Machine.stFillerModule.iq_astSubModuleAxis[CST_Outlet05].iq_stStatus.q_stMainAxisStatus.q_xTorqueError;
		MC_InputOutput.Network.Filler.Exceptions.Outlet05TrackException				:= VAR_Machine.stFillerModule.iq_astSubModuleAxis[CST_Outlet05].iq_stStatus.q_stMainAxisStatus.q_xLagError;
		MC_InputOutput.Network.Filler.Exceptions.Outlet05HomeException				:= NOT VAR_Machine.stFillerModule.iq_astSubModuleAxis[CST_Outlet05].iq_stStatus.q_stMainAxisStatus.q_xIsHomed AND
																						VAR_Machine.stFillerModule.iq_astSubModuleAxis[CST_Outlet05].iq_stStatus.q_stMainAxisStatus.q_xInitDone;
	END_IF

	IF VAR_Machine.stFillerModule.iq_astSubModuleAxis[CST_Outlet06].iq_stStatus.q_stMainAxisStatus.q_xAxisReal THEN
		IF NOT CFG_MC.Axes.Filler.Out[6].VelocityControl THEN
			MC_InputOutput.Network.Filler.Exceptions.Outlet06NotInOpException			:= NOT VAR_Machine.stFillerModule.iq_astSubModuleAxis[CST_Outlet06].iq_stStatus.q_stMainAxisStatus.iq_xOperational;
			MC_InputOutput.Network.Filler.Exceptions.Outlet06SafetyException			:= NOT MC_InputOutput.Safety.Filler.Commands.AxesDiag[CST_Outlet06].DI_NotErrFUNC;
		END_IF
		MC_InputOutput.Network.Filler.Exceptions.Outlet06DriveException 			:= VAR_Machine.stFillerModule.iq_astSubModuleAxis[CST_Outlet06].iq_stStatus.q_stMainAxisStatus.q_xError;
		MC_InputOutput.Network.Filler.Exceptions.Outlet06TorqueException			:= VAR_Machine.stFillerModule.iq_astSubModuleAxis[CST_Outlet06].iq_stStatus.q_stMainAxisStatus.q_xTorqueError;
		MC_InputOutput.Network.Filler.Exceptions.Outlet06TrackException 			:= VAR_Machine.stFillerModule.iq_astSubModuleAxis[CST_Outlet06].iq_stStatus.q_stMainAxisStatus.q_xLagError;
		MC_InputOutput.Network.Filler.Exceptions.Outlet06HomeException				:= NOT VAR_Machine.stFillerModule.iq_astSubModuleAxis[CST_Outlet06].iq_stStatus.q_stMainAxisStatus.q_xIsHomed AND
																						VAR_Machine.stFillerModule.iq_astSubModuleAxis[CST_Outlet06].iq_stStatus.q_stMainAxisStatus.q_xInitDone;
	END_IF
END_ACTION
